LIN {X 0,Y 457.388,Z 987.215,A -85,B 0,C 180,E1 20807.693,E2 20807.693} C_VEL
LIN {X 0,Y 456.712,Z 996.163,A -85,B 0,C 180,E1 20804.974,E2 20804.974} C_VEL
LIN {X 0,Y 456.27,Z 1003.644,A -85,B 0,C 180,E1 20802.148,E2 20802.148} C_VEL
LIN {X 0,Y 456.039,Z 1009.592,A -85,B 0,C 180,E1 20799.341,E2 20799.341} C_VEL
LIN {X 0,Y 455.943,Z 1013.795,A -85,B 0,C 180,E1 20796.551,E2 20796.551} C_VEL
LIN {X 0,Y 455.903,Z 1016.656,A -85,B 0,C 180,E1 20793.742,E2 20793.742} C_VEL
LIN {X 0,Y 455.893,Z 1017.826,A -85,B 0,C 180,E1 20791.009,E2 20791.009} C_VEL
LIN {X 0,Y 455.907,Z 1017.736,A -85,B 0,C 180,E1 20788.496,E2 20788.496} C_VEL
LIN {X 0,Y 455.909,Z 1016.072,A -85,B 0,C 180,E1 20785.602,E2 20785.602} C_VEL
LIN {X 0,Y 455.929,Z 1013.325,A -85,B 0,C 180,E1 20783.076,E2 20783.076} C_VEL
LIN {X 0,Y 456.047,Z 1008.599,A -85,B 0,C 180,E1 20780.158,E2 20780.158} C_VEL
LIN {X 0,Y 456.296,Z 1003.055,A -85,B 0,C 180,E1 20777.604,E2 20777.604} C_VEL
LIN {X 0,Y 456.792,Z 994.972,A -85,B 0,C 180,E1 20774.646,E2 20774.646} C_VEL
LIN {X 0,Y 457.469,Z 986.329,A -85,B 0,C 180,E1 20772.056,E2 20772.056} C_VEL
LIN {X 0,Y 458.569,Z 974.886,A -85,B 0,C 180,E1 20769.187,E2 20769.187} C_VEL
LIN {X 0,Y 460.023,Z 962.424,A -85,B 0,C 180,E1 20766.521,E2 20766.521} C_VEL
LIN {X 0,Y 461.834,Z 948.138,A -85,B 0,C 180,E1 20763.934,E2 20763.934} C_VEL
LIN {X 0,Y 464.101,Z 931.678,A -85,B 0,C 180,E1 20761.362,E2 20761.362} C_VEL
LIN {X 0,Y 466.447,Z 915.587,A -85,B 0,C 180,E1 20759.188,E2 20759.188} C_VEL
LIN {X 0,Y 468.959,Z 897.775,A -85,B 0,C 180,E1 20757.143,E2 20757.143} C_VEL
LIN {X 0,Y 471.666,Z 878.661,A -85,B 0,C 180,E1 20755.239,E2 20755.239} C_VEL
LIN {X 0,Y 474.239,Z 859.314,A -85,B 0,C 180,E1 20753.601,E2 20753.601} C_VEL
LIN {X 0,Y 477.014,Z 837.668,A -85,B 0,C 180,E1 20752.04,E2 20752.04} C_VEL
LIN {X 0,Y 479.232,Z 818.477,A -85,B 0,C 180,E1 20750.881,E2 20750.881} C_VEL
LIN {X 0,Y 481.541,Z 795.78,A -85,B 0,C 180,E1 20749.746,E2 20749.746} C_VEL
LIN {X 0,Y 483.409,Z 774.499,A -85,B 0,C 180,E1 20748.904,E2 20748.904} C_VEL
LIN {X 0,Y 485.034,Z 751.209,A -85,B 0,C 180,E1 20748.211,E2 20748.211} C_VEL
LIN {X 0,Y 486.068,Z 729.261,A -85,B 0,C 180,E1 20747.744,E2 20747.744} C_VEL
LIN {X 0,Y 491.465,Z 519.393,A -85,B 0,C 180,E1 20744.134,E2 20744.134} C_VEL
LIN {X 0,Y 493.764,Z 431.768,A -85,B 0,C 180,E1 20742.579,E2 20742.579} C_VEL
LIN {X 0,Y 480.7,Z 411.514,A -85,B 0,C 180,E1 20740.427,E2 20740.427} C_VEL
LIN {X 0,Y 467.612,Z 392.787,A -85,B 0,C 180,E1 20738.088,E2 20738.088} C_VEL
LIN {X 0,Y 463.575,Z 387.235,A -85,B 0,C 180,E1 20737.305,E2 20737.305} C_VEL
LIN {X 0,Y 460.808,Z 382.127,A -85,B 0,C 180,E1 20736.324,E2 20736.324} C_VEL
LIN {X 0,Y 458.868,Z 378.314,A -85,B 0,C 180,E1 20735.575,E2 20735.575} C_VEL
LIN {X 0,Y 457.218,Z 375.201,A -85,B 0,C 180,E1 20734.919,E2 20734.919} C_VEL
LIN {X 0,Y 457.037,Z 374.285,A -85,B 0,C 180,E1 20734.666,E2 20734.666} C_VEL
LIN {X 0,Y 456.993,Z 374.082,A -85,B 0,C 180,E1 20731.087,E2 20731.087} C_VEL
LIN {X 0,Y 457.031,Z 374.12,A -85,B 0,C 180,E1 20727.632,E2 20727.632} C_VEL
LIN {X 0,Y 457.038,Z 374.112,A -85,B 0,C 180,E1 20724.01,E2 20724.01} C_VEL
LIN {X 0,Y 456.998,Z 374.114,A -85,B 0,C 180,E1 20720.491,E2 20720.491} C_VEL
LIN {X 0,Y 457.001,Z 374.12,A -85,B 0,C 180,E1 20716.786,E2 20716.786} C_VEL
LIN {X 0,Y 457.043,Z 374.118,A -85,B 0,C 180,E1 20713.243,E2 20713.243} C_VEL
LIN {X 0,Y 457.048,Z 374.113,A -85,B 0,C 180,E1 20709.57,E2 20709.57} C_VEL
LIN {X 0,Y 457.01,Z 374.116,A -85,B 0,C 180,E1 20706.028,E2 20706.028} C_VEL
LIN {X 0,Y 457.01,Z 374.11,A -85,B 0,C 180,E1 20702.382,E2 20702.382} C_VEL
LIN {X 0,Y 457.057,Z 374.107,A -85,B 0,C 180,E1 20698.871,E2 20698.871} C_VEL
LIN {X 0,Y 457.05,Z 374.108,A -85,B 0,C 180,E1 20695.231,E2 20695.231} C_VEL
LIN {X 0,Y 457.017,Z 374.108,A -85,B 0,C 180,E1 20691.697,E2 20691.697} C_VEL
LIN {X 0,Y 457.021,Z 374.113,A -85,B 0,C 180,E1 20687.912,E2 20687.912} C_VEL
LIN {X 0,Y 457.061,Z 374.111,A -85,B 0,C 180,E1 20684.39,E2 20684.39} C_VEL
LIN {X 0,Y 457.067,Z 374.11,A -85,B 0,C 180,E1 20680.711,E2 20680.711} C_VEL
LIN {X 0,Y 457.039,Z 374.113,A -85,B 0,C 180,E1 20677.06,E2 20677.06} C_VEL
LIN {X 0,Y 457.03,Z 374.116,A -85,B 0,C 180,E1 20673.353,E2 20673.353} C_VEL
LIN {X 0,Y 457.054,Z 374.113,A -85,B 0,C 180,E1 20669.769,E2 20669.769} C_VEL
LIN {X 0,Y 457.078,Z 374.109,A -85,B 0,C 180,E1 20666.095,E2 20666.095} C_VEL
LIN {X 0,Y 457.064,Z 374.108,A -85,B 0,C 180,E1 20662.354,E2 20662.354} C_VEL
LIN {X 0,Y 457.038,Z 374.108,A -85,B 0,C 180,E1 20658.805,E2 20658.805} C_VEL
LIN {X 0,Y 457.046,Z 374.112,A -85,B 0,C 180,E1 20655.039,E2 20655.039} C_VEL
LIN {X 0,Y 457.074,Z 374.11,A -85,B 0,C 180,E1 20651.341,E2 20651.341} C_VEL
LIN {X 0,Y 457.075,Z 374.106,A -85,B 0,C 180,E1 20647.606,E2 20647.606} C_VEL
LIN {X 0,Y 457.064,Z 374.081,A -85,B 0,C 180,E1 20643.9,E2 20643.9} C_VEL
LIN {X 0,Y 457.046,Z 374.093,A -85,B 0,C 180,E1 20640.204,E2 20640.204} C_VEL
LIN {X 0,Y 457.054,Z 374.104,A -85,B 0,C 180,E1 20636.499,E2 20636.499} C_VEL
LIN {X 0,Y 457.104,Z 374.331,A -85,B 0,C 180,E1 20635.59,E2 20635.59} C_VEL
LIN {X 0,Y 457.483,Z 375.807,A -85,B 0,C 180,E1 20635.33,E2 20635.33} C_VEL
LIN {X 0,Y 459.463,Z 378.86,A -85,B 0,C 180,E1 20634.917,E2 20634.917} C_VEL
LIN {X 0,Y 461.42,Z 380.68,A -85,B 0,C 180,E1 20634.555,E2 20634.555} C_VEL
LIN {X 0,Y 463.984,Z 384.517,A -85,B 0,C 180,E1 20634.054,E2 20634.054} C_VEL
LIN {X 0,Y 465.802,Z 386.508,A -85,B 0,C 180,E1 20633.723,E2 20633.723} C_VEL
LIN {X 0,Y 469.108,Z 390.836,A -85,B 0,C 180,E1 20633.116,E2 20633.116} C_VEL
LIN {X 0,Y 478.42,Z 403.372,A -85,B 0,C 180,E1 20631.472,E2 20631.472} C_VEL
LIN {X 0,Y 488.967,Z 418.075,A -85,B 0,C 180,E1 20629.724,E2 20629.724} C_VEL
LIN {X 0,Y 490.028,Z 420.976,A -85,B 0,C 180,E1 20629.525,E2 20629.525} C_VEL
LIN {X 0,Y 490.141,Z 425.981,A -85,B 0,C 180,E1 20629.403,E2 20629.403} C_VEL
LIN {X 0,Y 487.747,Z 440.24,A -85,B 0,C 180,E1 20629.401,E2 20629.401} C_VEL
LIN {X 0,Y 487.657,Z 441.856,A -85,B 0,C 180,E1 20629.377,E2 20629.377} C_VEL
LIN {X 0,Y 481.671,Z 650.549,A -85,B 0,C 180,E1 20625.725,E2 20625.725} C_VEL
LIN {X 0,Y 479.794,Z 714.191,A -85,B 0,C 180,E1 20624.597,E2 20624.597} C_VEL
LIN {X 0,Y 478.39,Z 736.235,A -85,B 0,C 180,E1 20624.011,E2 20624.011} C_VEL
LIN {X 0,Y 476.654,Z 758.004,A -85,B 0,C 180,E1 20623.244,E2 20623.244} C_VEL
LIN {X 0,Y 474.492,Z 778.957,A -85,B 0,C 180,E1 20622.284,E2 20622.284} C_VEL
LIN {X 0,Y 472.041,Z 800.065,A -85,B 0,C 180,E1 20621.109,E2 20621.109} C_VEL
LIN {X 0,Y 469.256,Z 820.947,A -85,B 0,C 180,E1 20619.686,E2 20619.686} C_VEL
LIN {X 0,Y 466.204,Z 842.112,A -85,B 0,C 180,E1 20617.968,E2 20617.968} C_VEL
LIN {X 0,Y 463.242,Z 861.264,A -85,B 0,C 180,E1 20616.129,E2 20616.129} C_VEL
LIN {X 0,Y 460.391,Z 879.229,A -85,B 0,C 180,E1 20614.106,E2 20614.106} C_VEL
LIN {X 0,Y 457.653,Z 896.341,A -85,B 0,C 180,E1 20611.874,E2 20611.874} C_VEL
LIN {X 0,Y 455.123,Z 912.905,A -85,B 0,C 180,E1 20609.367,E2 20609.367} C_VEL
LIN {X 0,Y 452.991,Z 928.049,A -85,B 0,C 180,E1 20606.706,E2 20606.706} C_VEL
LIN {X 0,Y 451.232,Z 941.671,A -85,B 0,C 180,E1 20603.891,E2 20603.891} C_VEL
LIN {X 0,Y 449.972,Z 952.813,A -85,B 0,C 180,E1 20601.177,E2 20601.177} C_VEL
LIN {X 0,Y 449.049,Z 962.76,A -85,B 0,C 180,E1 20598.306,E2 20598.306} C_VEL
LIN {X 0,Y 448.483,Z 970.738,A -85,B 0,C 180,E1 20595.537,E2 20595.537} C_VEL
LIN {X 0,Y 448.133,Z 977.415,A -85,B 0,C 180,E1 20592.601,E2 20592.601} C_VEL
LIN {X 0,Y 447.981,Z 982.493,A -85,B 0,C 180,E1 20589.621,E2 20589.621} C_VEL
LIN {X 0,Y 447.897,Z 985.857,A -85,B 0,C 180,E1 20586.723,E2 20586.723} C_VEL
LIN {X 0,Y 447.888,Z 987.555,A -85,B 0,C 180,E1 20584.049,E2 20584.049} C_VEL
LIN {X 0,Y 447.91,Z 987.88,A -85,B 0,C 180,E1 20581.169,E2 20581.169} C_VEL
LIN {X 0,Y 447.909,Z 986.719,A -85,B 0,C 180,E1 20578.267,E2 20578.267} C_VEL
LIN {X 0,Y 447.936,Z 984.049,A -85,B 0,C 180,E1 20575.454,E2 20575.454} C_VEL
LIN {X 0,Y 448.052,Z 979.57,A -85,B 0,C 180,E1 20572.464,E2 20572.464} C_VEL
LIN {X 0,Y 448.304,Z 973.504,A -85,B 0,C 180,E1 20569.512,E2 20569.512} C_VEL
LIN {X 0,Y 448.79,Z 966.054,A -85,B 0,C 180,E1 20566.667,E2 20566.667} C_VEL
LIN {X 0,Y 449.539,Z 957.052,A -85,B 0,C 180,E1 20563.89,E2 20563.89} C_VEL
LIN {X 0,Y 450.685,Z 946.027,A -85,B 0,C 180,E1 20561.032,E2 20561.032} C_VEL
LIN {X 0,Y 452.23,Z 933.522,A -85,B 0,C 180,E1 20558.286,E2 20558.286} C_VEL
LIN {X 0,Y 454.16,Z 919.615,A -85,B 0,C 180,E1 20555.668,E2 20555.668} C_VEL
LIN {X 0,Y 456.632,Z 903.032,A -85,B 0,C 180,E1 20553.001,E2 20553.001} C_VEL
LIN {X 0,Y 459.267,Z 886.37,A -85,B 0,C 180,E1 20550.686,E2 20550.686} C_VEL
LIN {X 0,Y 462.142,Z 868.444,A -85,B 0,C 180,E1 20548.547,E2 20548.547} C_VEL
LIN {X 0,Y 465.202,Z 848.965,A -85,B 0,C 180,E1 20546.555,E2 20546.555} C_VEL
LIN {X 0,Y 468.061,Z 829.672,A -85,B 0,C 180,E1 20544.887,E2 20544.887} C_VEL
LIN {X 0,Y 471.021,Z 808.171,A -85,B 0,C 180,E1 20543.322,E2 20543.322} C_VEL
LIN {X 0,Y 473.405,Z 788.946,A -85,B 0,C 180,E1 20542.149,E2 20542.149} C_VEL
LIN {X 0,Y 475.719,Z 767.129,A -85,B 0,C 180,E1 20541.058,E2 20541.058} C_VEL
LIN {X 0,Y 477.718,Z 745.192,A -85,B 0,C 180,E1 20540.186,E2 20540.186} C_VEL
LIN {X 0,Y 479.228,Z 723.054,A -85,B 0,C 180,E1 20539.533,E2 20539.533} C_VEL
LIN {X 0,Y 480.309,Z 699.745,A -85,B 0,C 180,E1 20539.041,E2 20539.041} C_VEL
LIN {X 0,Y 486.203,Z 492.347,A -85,B 0,C 180,E1 20535.419,E2 20535.419} C_VEL
LIN {X 0,Y 488.107,Z 428.574,A -85,B 0,C 180,E1 20534.261,E2 20534.261} C_VEL
LIN {X 0,Y 476.707,Z 412.081,A -85,B 0,C 180,E1 20532.292,E2 20532.292} C_VEL
LIN {X 0,Y 468.825,Z 401.437,A -85,B 0,C 180,E1 20530.818,E2 20530.818} C_VEL
LIN {X 0,Y 465.589,Z 397.118,A -85,B 0,C 180,E1 20530.174,E2 20530.174} C_VEL
LIN {X 0,Y 461.719,Z 392.083,A -85,B 0,C 180,E1 20529.379,E2 20529.379} C_VEL
LIN {X 0,Y 458.545,Z 387.858,A -85,B 0,C 180,E1 20528.701,E2 20528.701} C_VEL
LIN {X 0,Y 454.704,Z 383.417,A -85,B 0,C 180,E1 20527.852,E2 20527.852} C_VEL
LIN {X 0,Y 453.422,Z 381.236,A -85,B 0,C 180,E1 20527.54,E2 20527.54} C_VEL
LIN {X 0,Y 450.618,Z 378.846,A -85,B 0,C 180,E1 20526.914,E2 20526.914} C_VEL
LIN {X 0,Y 449.296,Z 376.022,A -85,B 0,C 180,E1 20526.517,E2 20526.517} C_VEL
LIN {X 0,Y 449.14,Z 375.145,A -85,B 0,C 180,E1 20526.135,E2 20526.135} C_VEL
LIN {X 0,Y 449.13,Z 375.094,A -85,B 0,C 180,E1 20522.297,E2 20522.297} C_VEL
LIN {X 0,Y 449.132,Z 375.104,A -85,B 0,C 180,E1 20518.597,E2 20518.597} C_VEL
LIN {X 0,Y 449.129,Z 375.095,A -85,B 0,C 180,E1 20514.892,E2 20514.892} C_VEL
LIN {X 0,Y 449.11,Z 375.105,A -85,B 0,C 180,E1 20511.293,E2 20511.293} C_VEL
LIN {X 0,Y 449.11,Z 375.104,A -85,B 0,C 180,E1 20507.529,E2 20507.529} C_VEL
LIN {X 0,Y 449.127,Z 375.105,A -85,B 0,C 180,E1 20503.843,E2 20503.843} C_VEL
LIN {X 0,Y 449.138,Z 375.096,A -85,B 0,C 180,E1 20500.087,E2 20500.087} C_VEL
LIN {X 0,Y 449.106,Z 375.095,A -85,B 0,C 180,E1 20496.515,E2 20496.515} C_VEL
LIN {X 0,Y 449.083,Z 375.101,A -85,B 0,C 180,E1 20492.844,E2 20492.844} C_VEL
LIN {X 0,Y 449.078,Z 375.107,A -85,B 0,C 180,E1 20489.049,E2 20489.049} C_VEL
LIN {X 0,Y 449.114,Z 375.407,A -85,B 0,C 180,E1 20486.905,E2 20486.905} C_VEL
LIN {X 0,Y 450.522,Z 378.747,A -85,B 0,C 180,E1 20486.105,E2 20486.105} C_VEL
LIN {X 0,Y 451.811,Z 380.403,A -85,B 0,C 180,E1 20485.638,E2 20485.638} C_VEL
LIN {X 0,Y 453.49,Z 383.976,A -85,B 0,C 180,E1 20484.869,E2 20484.869} C_VEL
LIN {X 0,Y 455.261,Z 386.404,A -85,B 0,C 180,E1 20484.409,E2 20484.409} C_VEL
LIN {X 0,Y 463.169,Z 397.175,A -85,B 0,C 180,E1 20482.695,E2 20482.695} C_VEL
LIN {X 0,Y 472.136,Z 410.094,A -85,B 0,C 180,E1 20480.91,E2 20480.91} C_VEL
LIN {X 0,Y 482.787,Z 426.603,A -85,B 0,C 180,E1 20478.966,E2 20478.966} C_VEL
LIN {X 0,Y 488.335,Z 435.911,A -85,B 0,C 180,E1 20478.017,E2 20478.017} C_VEL
LIN {X 0,Y 482.34,Z 638.533,A -85,B 0,C 180,E1 20474.438,E2 20474.438} C_VEL
LIN {X 0,Y 479.526,Z 739.163,A -85,B 0,C 180,E1 20472.679,E2 20472.679} C_VEL
LIN {X 0,Y 478.027,Z 762.384,A -85,B 0,C 180,E1 20472.086,E2 20472.086} C_VEL
LIN {X 0,Y 476.191,Z 785.264,A -85,B 0,C 180,E1 20471.29,E2 20471.29} C_VEL
LIN {X 0,Y 474.079,Z 805.95,A -85,B 0,C 180,E1 20470.355,E2 20470.355} C_VEL
LIN {X 0,Y 471.772,Z 826.309,A -85,B 0,C 180,E1 20469.247,E2 20469.247} C_VEL
LIN {X 0,Y 469.076,Z 847.044,A -85,B 0,C 180,E1 20467.874,E2 20467.874} C_VEL
LIN {X 0,Y 466.295,Z 867.604,A -85,B 0,C 180,E1 20466.27,E2 20466.27} C_VEL
LIN {X 0,Y 463.565,Z 886.173,A -85,B 0,C 180,E1 20464.562,E2 20464.562} C_VEL
LIN {X 0,Y 460.689,Z 905.523,A -85,B 0,C 180,E1 20462.503,E2 20462.503} C_VEL
LIN {X 0,Y 458.231,Z 921.98,A -85,B 0,C 180,E1 20460.472,E2 20460.472} C_VEL
LIN {X 0,Y 455.93,Z 937.422,A -85,B 0,C 180,E1 20458.277,E2 20458.277} C_VEL
LIN {X 0,Y 453.922,Z 951.172,A -85,B 0,C 180,E1 20456.001,E2 20456.001} C_VEL
LIN {X 0,Y 452.029,Z 965.155,A -85,B 0,C 180,E1 20453.328,E2 20453.328} C_VEL
LIN {X 0,Y 450.586,Z 977.139,A -85,B 0,C 180,E1 20450.663,E2 20450.663} C_VEL
LIN {X 0,Y 449.491,Z 987.673,A -85,B 0,C 180,E1 20447.88,E2 20447.88} C_VEL
LIN {X 0,Y 448.769,Z 996.559,A -85,B 0,C 180,E1 20445.114,E2 20445.114} C_VEL
LIN {X 0,Y 448.305,Z 1003.687,A -85,B 0,C 180,E1 20442.348,E2 20442.348} C_VEL
LIN {X 0,Y 448.046,Z 1009.649,A -85,B 0,C 180,E1 20439.475,E2 20439.475} C_VEL
LIN {X 0,Y 447.94,Z 1013.828,A -85,B 0,C 180,E1 20436.642,E2 20436.642} C_VEL
LIN {X 0,Y 447.905,Z 1016.677,A -85,B 0,C 180,E1 20433.775,E2 20433.775} C_VEL
LIN {X 0,Y 447.894,Z 1017.826,A -85,B 0,C 180,E1 20431.027,E2 20431.027} C_VEL
LIN {X 0,Y 447.907,Z 1017.736,A -85,B 0,C 180,E1 20428.469,E2 20428.469} C_VEL
LIN {X 0,Y 447.908,Z 1016.072,A -85,B 0,C 180,E1 20425.523,E2 20425.523} C_VEL
LIN {X 0,Y 447.93,Z 1013.325,A -85,B 0,C 180,E1 20422.952,E2 20422.952} C_VEL
LIN {X 0,Y 448.063,Z 1008.599,A -85,B 0,C 180,E1 20419.981,E2 20419.981} C_VEL
LIN {X 0,Y 448.338,Z 1003.055,A -85,B 0,C 180,E1 20417.38,E2 20417.38} C_VEL
LIN {X 0,Y 448.879,Z 994.971,A -85,B 0,C 180,E1 20414.369,E2 20414.369} C_VEL
LIN {X 0,Y 449.628,Z 986.285,A -85,B 0,C 180,E1 20411.719,E2 20411.719} C_VEL
LIN {X 0,Y 450.826,Z 974.885,A -85,B 0,C 180,E1 20408.812,E2 20408.812} C_VEL
LIN {X 0,Y 452.363,Z 962.648,A -85,B 0,C 180,E1 20406.146,E2 20406.146} C_VEL
LIN {X 0,Y 454.245,Z 948.907,A -85,B 0,C 180,E1 20403.606,E2 20403.606} C_VEL
LIN {X 0,Y 456.476,Z 933.886,A -85,B 0,C 180,E1 20401.181,E2 20401.181} C_VEL
LIN {X 0,Y 458.78,Z 918.361,A -85,B 0,C 180,E1 20399.053,E2 20399.053} C_VEL
LIN {X 0,Y 461.578,Z 899.875,A -85,B 0,C 180,E1 20396.847,E2 20396.847} C_VEL
LIN {X 0,Y 464.205,Z 882.408,A -85,B 0,C 180,E1 20395.051,E2 20395.051} C_VEL
LIN {X 0,Y 467.116,Z 862.195,A -85,B 0,C 180,E1 20393.26,E2 20393.26} C_VEL
LIN {X 0,Y 469.763,Z 843.056,A -85,B 0,C 180,E1 20391.814,E2 20391.814} C_VEL
LIN {X 0,Y 472.361,Z 822.483,A -85,B 0,C 180,E1 20390.507,E2 20390.507} C_VEL
LIN {X 0,Y 474.434,Z 804.256,A -85,B 0,C 180,E1 20389.533,E2 20389.533} C_VEL
LIN {X 0,Y 476.688,Z 781.174,A -85,B 0,C 180,E1 20388.527,E2 20388.527} C_VEL
LIN {X 0,Y 478.399,Z 759.67,A -85,B 0,C 180,E1 20387.805,E2 20387.805} C_VEL
LIN {X 0,Y 479.828,Z 735.636,A -85,B 0,C 180,E1 20387.232,E2 20387.232} C_VEL
LIN {X 0,Y 485.614,Z 527.459,A -85,B 0,C 180,E1 20383.602,E2 20383.602} C_VEL
LIN {X 0,Y 488.182,Z 435.454,A -85,B 0,C 180,E1 20381.953,E2 20381.953} C_VEL
LIN {X 0,Y 476.406,Z 417.107,A -85,B 0,C 180,E1 20379.957,E2 20379.957} C_VEL
LIN {X 0,Y 463.992,Z 399.176,A -85,B 0,C 180,E1 20377.694,E2 20377.694} C_VEL
LIN {X 0,Y 455.028,Z 386.96,A -85,B 0,C 180,E1 20375.922,E2 20375.922} C_VEL
LIN {X 0,Y 453.441,Z 383.956,A -85,B 0,C 180,E1 20375.337,E2 20375.337} C_VEL
LIN {X 0,Y 450.759,Z 379.042,A -85,B 0,C 180,E1 20374.292,E2 20374.292} C_VEL
LIN {X 0,Y 449.099,Z 375.317,A -85,B 0,C 180,E1 20373.456,E2 20373.456} C_VEL
LIN {X 0,Y 449.116,Z 375.058,A -85,B 0,C 180,E1 20370.012,E2 20370.012} C_VEL
LIN {X 0,Y 449.067,Z 375.101,A -85,B 0,C 180,E1 20366.442,E2 20366.442} C_VEL
LIN {X 0,Y 449.056,Z 375.103,A -85,B 0,C 180,E1 20362.794,E2 20362.794} C_VEL
LIN {X 0,Y 449.082,Z 375.11,A -85,B 0,C 180,E1 20359.239,E2 20359.239} C_VEL
LIN {X 0,Y 449.12,Z 375.098,A -85,B 0,C 180,E1 20355.494,E2 20355.494} C_VEL
LIN {X 0,Y 449.091,Z 375.099,A -85,B 0,C 180,E1 20351.819,E2 20351.819} C_VEL
LIN {X 0,Y 449.065,Z 375.1,A -85,B 0,C 180,E1 20348.192,E2 20348.192} C_VEL
LIN {X 0,Y 449.073,Z 375.107,A -85,B 0,C 180,E1 20344.469,E2 20344.469} C_VEL
LIN {X 0,Y 449.113,Z 375.106,A -85,B 0,C 180,E1 20340.892,E2 20340.892} C_VEL
LIN {X 0,Y 449.119,Z 375.106,A -85,B 0,C 180,E1 20337.192,E2 20337.192} C_VEL
LIN {X 0,Y 449.082,Z 375.108,A -85,B 0,C 180,E1 20333.608,E2 20333.608} C_VEL
LIN {X 0,Y 449.08,Z 375.107,A -85,B 0,C 180,E1 20329.869,E2 20329.869} C_VEL
LIN {X 0,Y 449.101,Z 375.102,A -85,B 0,C 180,E1 20326.218,E2 20326.218} C_VEL
LIN {X 0,Y 449.133,Z 375.097,A -85,B 0,C 180,E1 20322.643,E2 20322.643} C_VEL
LIN {X 0,Y 449.104,Z 375.101,A -85,B 0,C 180,E1 20318.995,E2 20318.995} C_VEL
LIN {X 0,Y 449.088,Z 375.101,A -85,B 0,C 180,E1 20315.396,E2 20315.396} C_VEL
LIN {X 0,Y 449.102,Z 375.093,A -85,B 0,C 180,E1 20311.691,E2 20311.691} C_VEL
LIN {X 0,Y 449.14,Z 375.093,A -85,B 0,C 180,E1 20308.156,E2 20308.156} C_VEL
LIN {X 0,Y 449.118,Z 375.097,A -85,B 0,C 180,E1 20304.474,E2 20304.474} C_VEL
LIN {X 0,Y 449.099,Z 375.103,A -85,B 0,C 180,E1 20300.776,E2 20300.776} C_VEL
LIN {X 0,Y 449.104,Z 375.104,A -85,B 0,C 180,E1 20297.057,E2 20297.057} C_VEL
LIN {X 0,Y 449.131,Z 375.092,A -85,B 0,C 180,E1 20293.456,E2 20293.456} C_VEL
LIN {X 0,Y 449.139,Z 375.096,A -85,B 0,C 180,E1 20289.704,E2 20289.704} C_VEL
LIN {X 0,Y 449.124,Z 375.102,A -85,B 0,C 180,E1 20285.989,E2 20285.989} C_VEL
LIN {X 0,Y 449.109,Z 375.089,A -85,B 0,C 180,E1 20282.291,E2 20282.291} C_VEL
LIN {X 0,Y 449.114,Z 375.072,A -85,B 0,C 180,E1 20278.592,E2 20278.592} C_VEL
LIN {X 0,Y 449.161,Z 375.309,A -85,B 0,C 180,E1 20276.931,E2 20276.931} C_VEL
LIN {X 0,Y 449.492,Z 376.701,A -85,B 0,C 180,E1 20276.669,E2 20276.669} C_VEL
LIN {X 0,Y 451.275,Z 379.636,A -85,B 0,C 180,E1 20276.273,E2 20276.273} C_VEL
LIN {X 0,Y 453.6,Z 381.672,A -85,B 0,C 180,E1 20275.818,E2 20275.818} C_VEL
LIN {X 0,Y 456.122,Z 385.504,A -85,B 0,C 180,E1 20275.293,E2 20275.293} C_VEL
LIN {X 0,Y 458.035,Z 387.55,A -85,B 0,C 180,E1 20274.925,E2 20274.925} C_VEL
LIN {X 0,Y 461.288,Z 391.848,A -85,B 0,C 180,E1 20274.293,E2 20274.293} C_VEL
LIN {X 0,Y 471.105,Z 404.838,A -85,B 0,C 180,E1 20272.485,E2 20272.485} C_VEL
LIN {X 0,Y 482.014,Z 419.923,A -85,B 0,C 180,E1 20270.601,E2 20270.601} C_VEL
LIN {X 0,Y 488.05,Z 428.946,A -85,B 0,C 180,E1 20269.606,E2 20269.606} C_VEL
LIN {X 0,Y 487.657,Z 441.856,A -85,B 0,C 180,E1 20269.377,E2 20269.377} C_VEL
LIN {X 0,Y 486.774,Z 449.554,A -85,B 0,C 180,E1 20269.324,E2 20269.324} C_VEL
LIN {X 0,Y 481.871,Z 470.179,A -85,B 0,C 180,E1 20269.506,E2 20269.506} C_VEL
LIN {X 0,Y 481.138,Z 476.789,A -85,B 0,C 180,E1 20269.456,E2 20269.456} C_VEL
LIN {X 0,Y 474.9,Z 685.168,A -85,B 0,C 180,E1 20265.786,E2 20265.786} C_VEL
LIN {X 0,Y 473.681,Z 717.796,A -85,B 0,C 180,E1 20265.165,E2 20265.165} C_VEL
LIN {X 0,Y 472.297,Z 738.069,A -85,B 0,C 180,E1 20264.607,E2 20264.607} C_VEL
LIN {X 0,Y 470.299,Z 760.875,A -85,B 0,C 180,E1 20263.771,E2 20263.771} C_VEL
LIN {X 0,Y 468.121,Z 780.902,A -85,B 0,C 180,E1 20262.83,E2 20262.83} C_VEL
LIN {X 0,Y 465.416,Z 802.513,A -85,B 0,C 180,E1 20261.59,E2 20261.59} C_VEL
LIN {X 0,Y 462.723,Z 821.616,A -85,B 0,C 180,E1 20260.265,E2 20260.265} C_VEL
LIN {X 0,Y 459.578,Z 842.279,A -85,B 0,C 180,E1 20258.566,E2 20258.566} C_VEL
LIN {X 0,Y 456.472,Z 861.304,A -85,B 0,C 180,E1 20256.726,E2 20256.726} C_VEL
LIN {X 0,Y 453.427,Z 879.309,A -85,B 0,C 180,E1 20254.676,E2 20254.676} C_VEL
LIN {X 0,Y 450.51,Z 896.471,A -85,B 0,C 180,E1 20252.413,E2 20252.413} C_VEL
LIN {X 0,Y 447.908,Z 912.218,A -85,B 0,C 180,E1 20249.996,E2 20249.996} C_VEL
LIN {X 0,Y 445.447,Z 927.997,A -85,B 0,C 180,E1 20247.166,E2 20247.166} C_VEL
LIN {X 0,Y 443.6,Z 941.026,A -85,B 0,C 180,E1 20244.434,E2 20244.434} C_VEL
LIN {X 0,Y 442.226,Z 952.261,A -85,B 0,C 180,E1 20241.676,E2 20241.676} C_VEL
LIN {X 0,Y 441.211,Z 962.3,A -85,B 0,C 180,E1 20238.758,E2 20238.758} C_VEL
LIN {X 0,Y 440.547,Z 970.685,A -85,B 0,C 180,E1 20235.808,E2 20235.808} C_VEL
LIN {X 0,Y 440.154,Z 977.362,A -85,B 0,C 180,E1 20232.82,E2 20232.82} C_VEL
LIN {X 0,Y 439.984,Z 982.422,A -85,B 0,C 180,E1 20229.809,E2 20229.809} C_VEL
LIN {X 0,Y 439.904,Z 985.83,A -85,B 0,C 180,E1 20226.842,E2 20226.842} C_VEL
LIN {X 0,Y 439.889,Z 987.538,A -85,B 0,C 180,E1 20224.122,E2 20224.122} C_VEL
LIN {X 0,Y 439.909,Z 987.885,A -85,B 0,C 180,E1 20221.19,E2 20221.19} C_VEL
LIN {X 0,Y 439.909,Z 986.816,A -85,B 0,C 180,E1 20218.326,E2 20218.326} C_VEL
LIN {X 0,Y 439.941,Z 984.072,A -85,B 0,C 180,E1 20215.359,E2 20215.359} C_VEL
LIN {X 0,Y 440.064,Z 979.622,A -85,B 0,C 180,E1 20212.321,E2 20212.321} C_VEL
LIN {X 0,Y 440.342,Z 973.597,A -85,B 0,C 180,E1 20209.324,E2 20209.324} C_VEL
LIN {X 0,Y 440.871,Z 966.121,A -85,B 0,C 180,E1 20206.41,E2 20206.41} C_VEL
LIN {X 0,Y 441.691,Z 957.124,A -85,B 0,C 180,E1 20203.579,E2 20203.579} C_VEL
LIN {X 0,Y 442.936,Z 946.099,A -85,B 0,C 180,E1 20200.667,E2 20200.667} C_VEL
LIN {X 0,Y 444.605,Z 933.597,A -85,B 0,C 180,E1 20197.871,E2 20197.871} C_VEL
LIN {X 0,Y 446.783,Z 919.178,A -85,B 0,C 180,E1 20195.11,E2 20195.11} C_VEL
LIN {X 0,Y 449.385,Z 903.427,A -85,B 0,C 180,E1 20192.511,E2 20192.511} C_VEL
LIN {X 0,Y 452.243,Z 886.493,A -85,B 0,C 180,E1 20190.124,E2 20190.124} C_VEL
LIN {X 0,Y 455.245,Z 868.873,A -85,B 0,C 180,E1 20188,E2 20188} C_VEL
LIN {X 0,Y 458.349,Z 850.337,A -85,B 0,C 180,E1 20186.069,E2 20186.069} C_VEL
LIN {X 0,Y 461.327,Z 831.286,A -85,B 0,C 180,E1 20184.393,E2 20184.393} C_VEL
LIN {X 0,Y 464.474,Z 809.871,A -85,B 0,C 180,E1 20182.798,E2 20182.798} C_VEL
LIN {X 0,Y 466.975,Z 790.764,A -85,B 0,C 180,E1 20181.61,E2 20181.61} C_VEL
LIN {X 0,Y 469.571,Z 767.813,A -85,B 0,C 180,E1 20180.439,E2 20180.439} C_VEL
LIN {X 0,Y 471.653,Z 746.082,A -85,B 0,C 180,E1 20179.565,E2 20179.565} C_VEL
LIN {X 0,Y 473.267,Z 723.764,A -85,B 0,C 180,E1 20178.897,E2 20178.897} C_VEL
LIN {X 0,Y 474.406,Z 700.716,A -85,B 0,C 180,E1 20178.402,E2 20178.402} C_VEL
LIN {X 0,Y 480.689,Z 494.451,A -85,B 0,C 180,E1 20174.756,E2 20174.756} C_VEL
LIN {X 0,Y 482.655,Z 432.375,A -85,B 0,C 180,E1 20173.615,E2 20173.615} C_VEL
LIN {X 0,Y 470.141,Z 414.244,A -85,B 0,C 180,E1 20171.35,E2 20171.35} C_VEL
LIN {X 0,Y 461.919,Z 403.31,A -85,B 0,C 180,E1 20169.721,E2 20169.721} C_VEL
LIN {X 0,Y 458.231,Z 398.502,A -85,B 0,C 180,E1 20168.944,E2 20168.944} C_VEL
LIN {X 0,Y 454.411,Z 393.527,A -85,B 0,C 180,E1 20168.096,E2 20168.096} C_VEL
LIN {X 0,Y 451.26,Z 389.54,A -85,B 0,C 180,E1 20167.368,E2 20167.368} C_VEL
LIN {X 0,Y 450.326,Z 388.205,A -85,B 0,C 180,E1 20167.143,E2 20167.143} C_VEL
LIN {X 0,Y 447.231,Z 385.014,A -85,B 0,C 180,E1 20166.419,E2 20166.419} C_VEL
LIN {X 0,Y 445.901,Z 382.445,A -85,B 0,C 180,E1 20166.05,E2 20166.05} C_VEL
LIN {X 0,Y 442.839,Z 380.034,A -85,B 0,C 180,E1 20165.294,E2 20165.294} C_VEL
LIN {X 0,Y 441.351,Z 376.979,A -85,B 0,C 180,E1 20164.809,E2 20164.809} C_VEL
LIN {X 0,Y 441.194,Z 376.113,A -85,B 0,C 180,E1 20164.302,E2 20164.302} C_VEL
LIN {X 0,Y 441.19,Z 376.084,A -85,B 0,C 180,E1 20160.52,E2 20160.52} C_VEL
LIN {X 0,Y 441.193,Z 376.081,A -85,B 0,C 180,E1 20156.753,E2 20156.753} C_VEL
LIN {X 0,Y 441.187,Z 376.093,A -85,B 0,C 180,E1 20152.971,E2 20152.971} C_VEL
LIN {X 0,Y 441.169,Z 376.092,A -85,B 0,C 180,E1 20149.29,E2 20149.29} C_VEL
LIN {X 0,Y 441.171,Z 376.095,A -85,B 0,C 180,E1 20145.564,E2 20145.564} C_VEL
LIN {X 0,Y 441.194,Z 376.092,A -85,B 0,C 180,E1 20141.913,E2 20141.913} C_VEL
LIN {X 0,Y 441.207,Z 376.088,A -85,B 0,C 180,E1 20138.043,E2 20138.043} C_VEL
LIN {X 0,Y 441.182,Z 376.085,A -85,B 0,C 180,E1 20134.207,E2 20134.207} C_VEL
LIN {X 0,Y 441.14,Z 376.086,A -85,B 0,C 180,E1 20130.688,E2 20130.688} C_VEL
LIN {X 0,Y 441.187,Z 376.396,A -85,B 0,C 180,E1 20128.492,E2 20128.492} C_VEL
LIN {X 0,Y 442.885,Z 380.136,A -85,B 0,C 180,E1 20127.5,E2 20127.5} C_VEL
LIN {X 0,Y 444.099,Z 381.894,A -85,B 0,C 180,E1 20126.986,E2 20126.986} C_VEL
LIN {X 0,Y 445.977,Z 385.156,A -85,B 0,C 180,E1 20126.298,E2 20126.298} C_VEL
LIN {X 0,Y 448.071,Z 387.766,A -85,B 0,C 180,E1 20125.783,E2 20125.783} C_VEL
LIN {X 0,Y 452.441,Z 393.552,A -85,B 0,C 180,E1 20124.737,E2 20124.737} C_VEL
LIN {X 0,Y 459.988,Z 403.937,A -85,B 0,C 180,E1 20123.058,E2 20123.058} C_VEL
LIN {X 0,Y 469.163,Z 417.43,A -85,B 0,C 180,E1 20121.184,E2 20121.184} C_VEL
LIN {X 0,Y 480.342,Z 435.102,A -85,B 0,C 180,E1 20119.108,E2 20119.108} C_VEL
LIN {X 0,Y 482.867,Z 439.645,A -85,B 0,C 180,E1 20118.658,E2 20118.658} C_VEL
LIN {X 0,Y 476.5,Z 641.209,A -85,B 0,C 180,E1 20115.059,E2 20115.059} C_VEL
LIN {X 0,Y 473.563,Z 739.133,A -85,B 0,C 180,E1 20113.324,E2 20113.324} C_VEL
LIN {X 0,Y 471.954,Z 762.476,A -85,B 0,C 180,E1 20112.722,E2 20112.722} C_VEL
LIN {X 0,Y 470,Z 785.356,A -85,B 0,C 180,E1 20111.915,E2 20111.915} C_VEL
LIN {X 0,Y 467.777,Z 805.975,A -85,B 0,C 180,E1 20110.973,E2 20110.973} C_VEL
LIN {X 0,Y 465.272,Z 826.811,A -85,B 0,C 180,E1 20109.824,E2 20109.824} C_VEL
LIN {X 0,Y 462.422,Z 847.413,A -85,B 0,C 180,E1 20108.439,E2 20108.439} C_VEL
LIN {X 0,Y 459.38,Z 868.407,A -85,B 0,C 180,E1 20106.769,E2 20106.769} C_VEL
LIN {X 0,Y 456.593,Z 886.36,A -85,B 0,C 180,E1 20105.091,E2 20105.091} C_VEL
LIN {X 0,Y 453.448,Z 906.097,A -85,B 0,C 180,E1 20102.949,E2 20102.949} C_VEL
LIN {X 0,Y 450.841,Z 922.566,A -85,B 0,C 180,E1 20100.878,E2 20100.878} C_VEL
LIN {X 0,Y 448.265,Z 938.906,A -85,B 0,C 180,E1 20098.501,E2 20098.501} C_VEL
LIN {X 0,Y 446.22,Z 952.711,A -85,B 0,C 180,E1 20096.198,E2 20096.198} C_VEL
LIN {X 0,Y 444.22,Z 966.423,A -85,B 0,C 180,E1 20093.481,E2 20093.481} C_VEL
LIN {X 0,Y 442.705,Z 978.253,A -85,B 0,C 180,E1 20090.769,E2 20090.769} C_VEL
LIN {X 0,Y 441.554,Z 988.589,A -85,B 0,C 180,E1 20087.94,E2 20087.94} C_VEL
LIN {X 0,Y 440.726,Z 997.983,A -85,B 0,C 180,E1 20084.858,E2 20084.858} C_VEL
LIN {X 0,Y 440.298,Z 1004.552,A -85,B 0,C 180,E1 20082.196,E2 20082.196} C_VEL
LIN {X 0,Y 440.042,Z 1010.423,A -85,B 0,C 180,E1 20079.156,E2 20079.156} C_VEL
LIN {X 0,Y 439.945,Z 1014.114,A -85,B 0,C 180,E1 20076.529,E2 20076.529} C_VEL
LIN {X 0,Y 439.892,Z 1016.846,A -85,B 0,C 180,E1 20073.522,E2 20073.522} C_VEL
LIN {X 0,Y 439.889,Z 1017.848,A -85,B 0,C 180,E1 20070.916,E2 20070.916} C_VEL
LIN {X 0,Y 439.909,Z 1017.66,A -85,B 0,C 180,E1 20068.05,E2 20068.05} C_VEL
LIN {X 0,Y 439.91,Z 1015.844,A -85,B 0,C 180,E1 20065.18,E2 20065.18} C_VEL
LIN {X 0,Y 439.967,Z 1012.686,A -85,B 0,C 180,E1 20062.299,E2 20062.299} C_VEL
LIN {X 0,Y 440.131,Z 1007.836,A -85,B 0,C 180,E1 20059.401,E2 20059.401} C_VEL
LIN {X 0,Y 440.487,Z 1001.528,A -85,B 0,C 180,E1 20056.484,E2 20056.484} C_VEL
LIN {X 0,Y 441.066,Z 993.755,A -85,B 0,C 180,E1 20053.679,E2 20053.679} C_VEL
LIN {X 0,Y 441.994,Z 984.459,A -85,B 0,C 180,E1 20050.857,E2 20050.857} C_VEL
LIN {X 0,Y 443.247,Z 973.736,A -85,B 0,C 180,E1 20048.154,E2 20048.154} C_VEL
LIN {X 0,Y 444.948,Z 961.269,A -85,B 0,C 180,E1 20045.441,E2 20045.441} C_VEL
LIN {X 0,Y 446.778,Z 948.862,A -85,B 0,C 180,E1 20043.129,E2 20043.129} C_VEL
LIN {X 0,Y 449.187,Z 933.255,A -85,B 0,C 180,E1 20040.623,E2 20040.623} C_VEL
LIN {X 0,Y 451.762,Z 916.967,A -85,B 0,C 180,E1 20038.369,E2 20038.369} C_VEL
LIN {X 0,Y 454.822,Z 898.07,A -85,B 0,C 180,E1 20036.115,E2 20036.115} C_VEL
LIN {X 0,Y 457.712,Z 879.987,A -85,B 0,C 180,E1 20034.25,E2 20034.25} C_VEL
LIN {X 0,Y 460.738,Z 860.144,A -85,B 0,C 180,E1 20032.51,E2 20032.51} C_VEL
LIN {X 0,Y 463.716,Z 839.852,A -85,B 0,C 180,E1 20030.986,E2 20030.986} C_VEL
LIN {X 0,Y 466.454,Z 818.606,A -85,B 0,C 180,E1 20029.665,E2 20029.665} C_VEL
LIN {X 0,Y 469.043,Z 796.277,A -85,B 0,C 180,E1 20028.522,E2 20028.522} C_VEL
LIN {X 0,Y 471.13,Z 775.083,A -85,B 0,C 180,E1 20027.665,E2 20027.665} C_VEL
LIN {X 0,Y 472.991,Z 751.564,A -85,B 0,C 180,E1 20026.945,E2 20026.945} C_VEL
LIN {X 0,Y 474.14,Z 729.857,A -85,B 0,C 180,E1 20026.471,E2 20026.471} C_VEL
LIN {X 0,Y 480.299,Z 519.471,A -85,B 0,C 180,E1 20022.774,E2 20022.774} C_VEL
LIN {X 0,Y 482.692,Z 439.246,A -85,B 0,C 180,E1 20021.319,E2 20021.319} C_VEL
LIN {X 0,Y 472.156,Z 422.69,A -85,B 0,C 180,E1 20019.48,E2 20019.48} C_VEL
LIN {X 0,Y 460.256,Z 405.397,A -85,B 0,C 180,E1 20017.268,E2 20017.268} C_VEL
LIN {X 0,Y 449.103,Z 390.229,A -85,B 0,C 180,E1 20015.018,E2 20015.018} C_VEL
LIN {X 0,Y 446.205,Z 385.768,A -85,B 0,C 180,E1 20014.302,E2 20014.302} C_VEL
LIN {X 0,Y 443.806,Z 381.453,A -85,B 0,C 180,E1 20013.347,E2 20013.347} C_VEL
LIN {X 0,Y 441.528,Z 377.731,A -85,B 0,C 180,E1 20012.458,E2 20012.458} C_VEL
LIN {X 0,Y 441.2,Z 376.276,A -85,B 0,C 180,E1 20012.094,E2 20012.094} C_VEL
LIN {X 0,Y 441.118,Z 376.074,A -85,B 0,C 180,E1 20008.707,E2 20008.707} C_VEL
LIN {X 0,Y 441.116,Z 376.102,A -85,B 0,C 180,E1 20004.935,E2 20004.935} C_VEL
LIN {X 0,Y 441.138,Z 376.094,A -85,B 0,C 180,E1 20001.262,E2 20001.262} C_VEL
LIN {X 0,Y 441.172,Z 376.086,A -85,B 0,C 180,E1 19997.543,E2 19997.543} C_VEL
LIN {X 0,Y 441.148,Z 376.09,A -85,B 0,C 180,E1 19993.901,E2 19993.901} C_VEL
LIN {X 0,Y 441.126,Z 376.097,A -85,B 0,C 180,E1 19990.315,E2 19990.315} C_VEL
LIN {X 0,Y 441.131,Z 376.095,A -85,B 0,C 180,E1 19986.507,E2 19986.507} C_VEL
LIN {X 0,Y 441.161,Z 376.086,A -85,B 0,C 180,E1 19982.858,E2 19982.858} C_VEL
LIN {X 0,Y 441.184,Z 376.084,A -85,B 0,C 180,E1 19979.22,E2 19979.22} C_VEL
LIN {X 0,Y 441.146,Z 376.088,A -85,B 0,C 180,E1 19975.58,E2 19975.58} C_VEL
LIN {X 0,Y 441.138,Z 376.085,A -85,B 0,C 180,E1 19971.921,E2 19971.921} C_VEL
LIN {X 0,Y 441.156,Z 376.087,A -85,B 0,C 180,E1 19968.23,E2 19968.23} C_VEL
LIN {X 0,Y 441.199,Z 376.083,A -85,B 0,C 180,E1 19964.624,E2 19964.624} C_VEL
LIN {X 0,Y 441.181,Z 376.086,A -85,B 0,C 180,E1 19960.815,E2 19960.815} C_VEL
LIN {X 0,Y 441.153,Z 376.091,A -85,B 0,C 180,E1 19957.196,E2 19957.196} C_VEL
LIN {X 0,Y 441.155,Z 376.093,A -85,B 0,C 180,E1 19953.481,E2 19953.481} C_VEL
LIN {X 0,Y 441.178,Z 376.092,A -85,B 0,C 180,E1 19949.792,E2 19949.792} C_VEL
LIN {X 0,Y 441.198,Z 376.086,A -85,B 0,C 180,E1 19946.031,E2 19946.031} C_VEL
LIN {X 0,Y 441.191,Z 376.083,A -85,B 0,C 180,E1 19942.263,E2 19942.263} C_VEL
LIN {X 0,Y 441.168,Z 376.084,A -85,B 0,C 180,E1 19938.563,E2 19938.563} C_VEL
LIN {X 0,Y 441.164,Z 376.091,A -85,B 0,C 180,E1 19934.81,E2 19934.81} C_VEL
LIN {X 0,Y 441.175,Z 376.089,A -85,B 0,C 180,E1 19931,E2 19931} C_VEL
LIN {X 0,Y 441.194,Z 376.084,A -85,B 0,C 180,E1 19927.301,E2 19927.301} C_VEL
LIN {X 0,Y 441.195,Z 376.054,A -85,B 0,C 180,E1 19923.489,E2 19923.489} C_VEL
LIN {X 0,Y 441.192,Z 376.058,A -85,B 0,C 180,E1 19919.75,E2 19919.75} C_VEL
LIN {X 0,Y 441.192,Z 376.214,A -85,B 0,C 180,E1 19918.413,E2 19918.413} C_VEL
LIN {X 0,Y 441.501,Z 377.549,A -85,B 0,C 180,E1 19918.097,E2 19918.097} C_VEL
LIN {X 0,Y 443.334,Z 380.596,A -85,B 0,C 180,E1 19917.655,E2 19917.655} C_VEL
LIN {X 0,Y 445.735,Z 382.707,A -85,B 0,C 180,E1 19917.164,E2 19917.164} C_VEL
LIN {X 0,Y 448.23,Z 386.518,A -85,B 0,C 180,E1 19916.618,E2 19916.618} C_VEL
LIN {X 0,Y 450.397,Z 388.731,A -85,B 0,C 180,E1 19916.179,E2 19916.179} C_VEL
LIN {X 0,Y 453.661,Z 393.015,A -85,B 0,C 180,E1 19915.506,E2 19915.506} C_VEL
LIN {X 0,Y 463.626,Z 406.113,A -85,B 0,C 180,E1 19913.571,E2 19913.571} C_VEL
LIN {X 0,Y 474.371,Z 420.762,A -85,B 0,C 180,E1 19911.639,E2 19911.639} C_VEL
LIN {X 0,Y 482.548,Z 432.768,A -85,B 0,C 180,E1 19910.242,E2 19910.242} C_VEL
LIN {X 0,Y 481.138,Z 476.789,A -85,B 0,C 180,E1 19909.456,E2 19909.456} C_VEL
LIN {X 0,Y 480.208,Z 484.487,A -85,B 0,C 180,E1 19909.407,E2 19909.407} C_VEL
LIN {X 0,Y 475.287,Z 505.1,A -85,B 0,C 180,E1 19909.592,E2 19909.592} C_VEL
LIN {X 0,Y 474.545,Z 511.706,A -85,B 0,C 180,E1 19909.542,E2 19909.542} C_VEL
LIN {X 0,Y 468.162,Z 711.488,A -85,B 0,C 180,E1 19905.976,E2 19905.976} C_VEL
LIN {X 0,Y 466.601,Z 735.251,A -85,B 0,C 180,E1 19905.365,E2 19905.365} C_VEL
LIN {X 0,Y 464.716,Z 756.98,A -85,B 0,C 180,E1 19904.599,E2 19904.599} C_VEL
LIN {X 0,Y 462.36,Z 778.198,A -85,B 0,C 180,E1 19903.629,E2 19903.629} C_VEL
LIN {X 0,Y 459.897,Z 797.56,A -85,B 0,C 180,E1 19902.553,E2 19902.553} C_VEL
LIN {X 0,Y 456.737,Z 819.042,A -85,B 0,C 180,E1 19901.103,E2 19901.103} C_VEL
LIN {X 0,Y 453.629,Z 838.871,A -85,B 0,C 180,E1 19899.511,E2 19899.511} C_VEL
LIN {X 0,Y 450.389,Z 857.664,A -85,B 0,C 180,E1 19897.714,E2 19897.714} C_VEL
LIN {X 0,Y 447.153,Z 875.853,A -85,B 0,C 180,E1 19895.702,E2 19895.702} C_VEL
LIN {X 0,Y 444.071,Z 892.964,A -85,B 0,C 180,E1 19893.481,E2 19893.481} C_VEL
LIN {X 0,Y 441.143,Z 909.197,A -85,B 0,C 180,E1 19891.035,E2 19891.035} C_VEL
LIN {X 0,Y 438.597,Z 923.997,A -85,B 0,C 180,E1 19888.429,E2 19888.429} C_VEL
LIN {X 0,Y 436.375,Z 938.082,A -85,B 0,C 180,E1 19885.528,E2 19885.528} C_VEL
LIN {X 0,Y 434.643,Z 950.72,A -85,B 0,C 180,E1 19882.462,E2 19882.462} C_VEL
LIN {X 0,Y 433.472,Z 961.032,A -85,B 0,C 180,E1 19879.497,E2 19879.497} C_VEL
LIN {X 0,Y 432.693,Z 969.551,A -85,B 0,C 180,E1 19876.5,E2 19876.5} C_VEL
LIN {X 0,Y 432.213,Z 976.469,A -85,B 0,C 180,E1 19873.465,E2 19873.465} C_VEL
LIN {X 0,Y 431.991,Z 981.627,A -85,B 0,C 180,E1 19870.528,E2 19870.528} C_VEL
LIN {X 0,Y 431.917,Z 985.134,A -85,B 0,C 180,E1 19867.685,E2 19867.685} C_VEL
LIN {X 0,Y 431.911,Z 987.25,A -85,B 0,C 180,E1 19864.786,E2 19864.786} C_VEL
LIN {X 0,Y 431.906,Z 987.984,A -85,B 0,C 180,E1 19861.816,E2 19861.816} C_VEL
LIN {X 0,Y 431.914,Z 987.155,A -85,B 0,C 180,E1 19858.917,E2 19858.917} C_VEL
LIN {X 0,Y 431.912,Z 984.814,A -85,B 0,C 180,E1 19855.926,E2 19855.926} C_VEL
LIN {X 0,Y 432.003,Z 981.321,A -85,B 0,C 180,E1 19853.166,E2 19853.166} C_VEL
LIN {X 0,Y 432.266,Z 975.915,A -85,B 0,C 180,E1 19850.17,E2 19850.17} C_VEL
LIN {X 0,Y 432.754,Z 968.702,A -85,B 0,C 180,E1 19847.09,E2 19847.09} C_VEL
LIN {X 0,Y 433.553,Z 960.159,A -85,B 0,C 180,E1 19844.145,E2 19844.145} C_VEL
LIN {X 0,Y 434.744,Z 949.907,A -85,B 0,C 180,E1 19841.227,E2 19841.227} C_VEL
LIN {X 0,Y 436.487,Z 937.277,A -85,B 0,C 180,E1 19838.206,E2 19838.206} C_VEL
LIN {X 0,Y 438.706,Z 923.476,A -85,B 0,C 180,E1 19835.373,E2 19835.373} C_VEL
LIN {X 0,Y 441.32,Z 908.376,A -85,B 0,C 180,E1 19832.728,E2 19832.728} C_VEL
LIN {X 0,Y 444.356,Z 891.566,A -85,B 0,C 180,E1 19830.222,E2 19830.222} C_VEL
LIN {X 0,Y 447.467,Z 874.588,A -85,B 0,C 180,E1 19828.036,E2 19828.036} C_VEL
LIN {X 0,Y 450.659,Z 856.495,A -85,B 0,C 180,E1 19826.059,E2 19826.059} C_VEL
LIN {X 0,Y 453.962,Z 837.102,A -85,B 0,C 180,E1 19824.235,E2 19824.235} C_VEL
LIN {X 0,Y 456.976,Z 817.991,A -85,B 0,C 180,E1 19822.718,E2 19822.718} C_VEL
LIN {X 0,Y 460.097,Z 796.384,A -85,B 0,C 180,E1 19821.28,E2 19821.28} C_VEL
LIN {X 0,Y 462.498,Z 777.435,A -85,B 0,C 180,E1 19820.236,E2 19820.236} C_VEL
LIN {X 0,Y 464.951,Z 754.313,A -85,B 0,C 180,E1 19819.206,E2 19819.206} C_VEL
LIN {X 0,Y 466.78,Z 732.967,A -85,B 0,C 180,E1 19818.472,E2 19818.472} C_VEL
LIN {X 0,Y 468.222,Z 709.434,A -85,B 0,C 180,E1 19817.899,E2 19817.899} C_VEL
LIN {X 0,Y 475.256,Z 496.565,A -85,B 0,C 180,E1 19814.078,E2 19814.078} C_VEL
LIN {X 0,Y 477.35,Z 436.488,A -85,B 0,C 180,E1 19812.969,E2 19812.969} C_VEL
LIN {X 0,Y 466.387,Z 420.405,A -85,B 0,C 180,E1 19810.916,E2 19810.916} C_VEL
LIN {X 0,Y 458.146,Z 409.3,A -85,B 0,C 180,E1 19809.231,E2 19809.231} C_VEL
LIN {X 0,Y 454.666,Z 404.739,A -85,B 0,C 180,E1 19808.473,E2 19808.473} C_VEL
LIN {X 0,Y 451.182,Z 400.154,A -85,B 0,C 180,E1 19807.674,E2 19807.674} C_VEL
LIN {X 0,Y 446.981,Z 394.841,A -85,B 0,C 180,E1 19806.676,E2 19806.676} C_VEL
LIN {X 0,Y 443.834,Z 390.995,A -85,B 0,C 180,E1 19805.884,E2 19805.884} C_VEL
LIN {X 0,Y 442.933,Z 389.52,A -85,B 0,C 180,E1 19805.636,E2 19805.636} C_VEL
LIN {X 0,Y 439.801,Z 386.532,A -85,B 0,C 180,E1 19804.826,E2 19804.826} C_VEL
LIN {X 0,Y 438.09,Z 383.493,A -85,B 0,C 180,E1 19804.32,E2 19804.32} C_VEL
LIN {X 0,Y 434.975,Z 381.129,A -85,B 0,C 180,E1 19803.46,E2 19803.46} C_VEL
LIN {X 0,Y 433.435,Z 378.048,A -85,B 0,C 180,E1 19802.91,E2 19802.91} C_VEL
LIN {X 0,Y 433.256,Z 377.11,A -85,B 0,C 180,E1 19802.381,E2 19802.381} C_VEL
LIN {X 0,Y 433.255,Z 377.082,A -85,B 0,C 180,E1 19798.546,E2 19798.546} C_VEL
LIN {X 0,Y 433.255,Z 377.069,A -85,B 0,C 180,E1 19794.704,E2 19794.704} C_VEL
LIN {X 0,Y 433.242,Z 377.081,A -85,B 0,C 180,E1 19790.972,E2 19790.972} C_VEL
LIN {X 0,Y 433.228,Z 377.083,A -85,B 0,C 180,E1 19787.2,E2 19787.2} C_VEL
LIN {X 0,Y 433.225,Z 377.083,A -85,B 0,C 180,E1 19783.371,E2 19783.371} C_VEL
LIN {X 0,Y 433.233,Z 377.071,A -85,B 0,C 180,E1 19779.605,E2 19779.605} C_VEL
LIN {X 0,Y 433.253,Z 377.07,A -85,B 0,C 180,E1 19775.891,E2 19775.891} C_VEL
LIN {X 0,Y 433.255,Z 377.083,A -85,B 0,C 180,E1 19772.065,E2 19772.065} C_VEL
LIN {X 0,Y 433.275,Z 377.415,A -85,B 0,C 180,E1 19770.255,E2 19770.255} C_VEL
LIN {X 0,Y 434.942,Z 381.152,A -85,B 0,C 180,E1 19769.161,E2 19769.161} C_VEL
LIN {X 0,Y 436.467,Z 383.151,A -85,B 0,C 180,E1 19768.552,E2 19768.552} C_VEL
LIN {X 0,Y 439.805,Z 387.572,A -85,B 0,C 180,E1 19767.592,E2 19767.592} C_VEL
LIN {X 0,Y 445.205,Z 394.708,A -85,B 0,C 180,E1 19766.154,E2 19766.154} C_VEL
LIN {X 0,Y 449.407,Z 400.317,A -85,B 0,C 180,E1 19765.126,E2 19765.126} C_VEL
LIN {X 0,Y 458.096,Z 412.422,A -85,B 0,C 180,E1 19763.154,E2 19763.154} C_VEL
LIN {X 0,Y 469.449,Z 429.806,A -85,B 0,C 180,E1 19760.829,E2 19760.829} C_VEL
LIN {X 0,Y 477.483,Z 443.285,A -85,B 0,C 180,E1 19759.317,E2 19759.317} C_VEL
LIN {X 0,Y 470.688,Z 644.968,A -85,B 0,C 180,E1 19755.676,E2 19755.676} C_VEL
LIN {X 0,Y 467.691,Z 738.695,A -85,B 0,C 180,E1 19753.996,E2 19753.996} C_VEL
LIN {X 0,Y 465.982,Z 762.147,A -85,B 0,C 180,E1 19753.388,E2 19753.388} C_VEL
LIN {X 0,Y 463.95,Z 784.701,A -85,B 0,C 180,E1 19752.589,E2 19752.589} C_VEL
LIN {X 0,Y 461.618,Z 805.26,A -85,B 0,C 180,E1 19751.647,E2 19751.647} C_VEL
LIN {X 0,Y 458.972,Z 826.241,A -85,B 0,C 180,E1 19750.483,E2 19750.483} C_VEL
LIN {X 0,Y 455.935,Z 847.01,A -85,B 0,C 180,E1 19749.076,E2 19749.076} C_VEL
LIN {X 0,Y 452.717,Z 867.896,A -85,B 0,C 180,E1 19747.402,E2 19747.402} C_VEL
LIN {X 0,Y 449.768,Z 885.871,A -85,B 0,C 180,E1 19745.704,E2 19745.704} C_VEL
LIN {X 0,Y 446.387,Z 905.792,A -85,B 0,C 180,E1 19743.517,E2 19743.517} C_VEL
LIN {X 0,Y 443.576,Z 922.519,A -85,B 0,C 180,E1 19741.382,E2 19741.382} C_VEL
LIN {X 0,Y 440.894,Z 938.399,A -85,B 0,C 180,E1 19739.036,E2 19739.036} C_VEL
LIN {X 0,Y 438.588,Z 953.131,A -85,B 0,C 180,E1 19736.543,E2 19736.543} C_VEL
LIN {X 0,Y 436.592,Z 966.402,A -85,B 0,C 180,E1 19733.917,E2 19733.917} C_VEL
LIN {X 0,Y 434.955,Z 978.244,A -85,B 0,C 180,E1 19731.159,E2 19731.159} C_VEL
LIN {X 0,Y 433.71,Z 988.588,A -85,B 0,C 180,E1 19728.276,E2 19728.276} C_VEL
LIN {X 0,Y 432.813,Z 997.982,A -85,B 0,C 180,E1 19725.136,E2 19725.136} C_VEL
LIN {X 0,Y 432.338,Z 1004.552,A -85,B 0,C 180,E1 19722.424,E2 19722.424} C_VEL
LIN {X 0,Y 432.051,Z 1010.423,A -85,B 0,C 180,E1 19719.326,E2 19719.326} C_VEL
LIN {X 0,Y 431.941,Z 1014.114,A -85,B 0,C 180,E1 19716.65,E2 19716.65} C_VEL
LIN {X 0,Y 431.895,Z 1016.846,A -85,B 0,C 180,E1 19713.588,E2 19713.588} C_VEL
LIN {X 0,Y 431.891,Z 1017.848,A -85,B 0,C 180,E1 19710.933,E2 19710.933} C_VEL
LIN {X 0,Y 431.907,Z 1017.69,A -85,B 0,C 180,E1 19708.147,E2 19708.147} C_VEL
LIN {X 0,Y 431.91,Z 1015.958,A -85,B 0,C 180,E1 19705.224,E2 19705.224} C_VEL
LIN {X 0,Y 431.947,Z 1013.165,A -85,B 0,C 180,E1 19702.556,E2 19702.556} C_VEL
LIN {X 0,Y 432.129,Z 1008.344,A -85,B 0,C 180,E1 19699.472,E2 19699.472} C_VEL
LIN {X 0,Y 432.462,Z 1002.683,A -85,B 0,C 180,E1 19696.742,E2 19696.742} C_VEL
LIN {X 0,Y 433.105,Z 994.564,A -85,B 0,C 180,E1 19693.646,E2 19693.646} C_VEL
LIN {X 0,Y 434.021,Z 985.867,A -85,B 0,C 180,E1 19690.911,E2 19690.911} C_VEL
LIN {X 0,Y 435.391,Z 974.881,A -85,B 0,C 180,E1 19688.023,E2 19688.023} C_VEL
LIN {X 0,Y 436.905,Z 964.222,A -85,B 0,C 180,E1 19685.618,E2 19685.618} C_VEL
LIN {X 0,Y 439.055,Z 950.09,A -85,B 0,C 180,E1 19682.911,E2 19682.911} C_VEL
LIN {X 0,Y 441.537,Z 935.032,A -85,B 0,C 180,E1 19680.407,E2 19680.407} C_VEL
LIN {X 0,Y 444.333,Z 918.324,A -85,B 0,C 180,E1 19678.031,E2 19678.031} C_VEL
LIN {X 0,Y 447.466,Z 900.292,A -85,B 0,C 180,E1 19675.806,E2 19675.806} C_VEL
LIN {X 0,Y 450.524,Z 882.137,A -85,B 0,C 180,E1 19673.884,E2 19673.884} C_VEL
LIN {X 0,Y 453.923,Z 861.381,A -85,B 0,C 180,E1 19672.007,E2 19672.007} C_VEL
LIN {X 0,Y 456.942,Z 841.935,A -85,B 0,C 180,E1 19670.513,E2 19670.513} C_VEL
LIN {X 0,Y 459.925,Z 820.441,A -85,B 0,C 180,E1 19669.136,E2 19669.136} C_VEL
LIN {X 0,Y 462.648,Z 798.755,A -85,B 0,C 180,E1 19667.985,E2 19667.985} C_VEL
LIN {X 0,Y 464.969,Z 776.396,A -85,B 0,C 180,E1 19667.059,E2 19667.059} C_VEL
LIN {X 0,Y 466.971,Z 752.989,A -85,B 0,C 180,E1 19666.32,E2 19666.32} C_VEL
LIN {X 0,Y 468.217,Z 731.065,A -85,B 0,C 180,E1 19665.829,E2 19665.829} C_VEL
LIN {X 0,Y 474.798,Z 520.557,A -85,B 0,C 180,E1 19662.087,E2 19662.087} C_VEL
LIN {X 0,Y 477.315,Z 443.079,A -85,B 0,C 180,E1 19660.679,E2 19660.679} C_VEL
LIN {X 0,Y 466.056,Z 425.409,A -85,B 0,C 180,E1 19658.652,E2 19658.652} C_VEL
LIN {X 0,Y 455.734,Z 410.548,A -85,B 0,C 180,E1 19656.676,E2 19656.676} C_VEL
LIN {X 0,Y 445.775,Z 396.779,A -85,B 0,C 180,E1 19654.608,E2 19654.608} C_VEL
LIN {X 0,Y 441.486,Z 391.088,A -85,B 0,C 180,E1 19653.662,E2 19653.662} C_VEL
LIN {X 0,Y 437.663,Z 386.025,A -85,B 0,C 180,E1 19652.781,E2 19652.781} C_VEL
LIN {X 0,Y 435.201,Z 381.422,A -85,B 0,C 180,E1 19651.743,E2 19651.743} C_VEL
LIN {X 0,Y 433.336,Z 377.917,A -85,B 0,C 180,E1 19650.881,E2 19650.881} C_VEL
LIN {X 0,Y 433.203,Z 377.127,A -85,B 0,C 180,E1 19650.515,E2 19650.515} C_VEL
LIN {X 0,Y 433.176,Z 377.082,A -85,B 0,C 180,E1 19646.898,E2 19646.898} C_VEL
LIN {X 0,Y 433.184,Z 377.077,A -85,B 0,C 180,E1 19643.103,E2 19643.103} C_VEL
LIN {X 0,Y 433.23,Z 377.08,A -85,B 0,C 180,E1 19639.551,E2 19639.551} C_VEL
LIN {X 0,Y 433.225,Z 377.082,A -85,B 0,C 180,E1 19635.782,E2 19635.782} C_VEL
LIN {X 0,Y 433.193,Z 377.079,A -85,B 0,C 180,E1 19632.124,E2 19632.124} C_VEL
LIN {X 0,Y 433.187,Z 377.076,A -85,B 0,C 180,E1 19628.361,E2 19628.361} C_VEL
LIN {X 0,Y 433.209,Z 377.079,A -85,B 0,C 180,E1 19624.766,E2 19624.766} C_VEL
LIN {X 0,Y 433.249,Z 377.078,A -85,B 0,C 180,E1 19621.057,E2 19621.057} C_VEL
LIN {X 0,Y 433.227,Z 377.083,A -85,B 0,C 180,E1 19617.354,E2 19617.354} C_VEL
LIN {X 0,Y 433.204,Z 377.086,A -85,B 0,C 180,E1 19613.639,E2 19613.639} C_VEL
LIN {X 0,Y 433.204,Z 377.085,A -85,B 0,C 180,E1 19609.897,E2 19609.897} C_VEL
LIN {X 0,Y 433.216,Z 377.08,A -85,B 0,C 180,E1 19606.111,E2 19606.111} C_VEL
LIN {X 0,Y 433.249,Z 377.071,A -85,B 0,C 180,E1 19602.402,E2 19602.402} C_VEL
LIN {X 0,Y 433.255,Z 377.07,A -85,B 0,C 180,E1 19598.615,E2 19598.615} C_VEL
LIN {X 0,Y 433.228,Z 377.073,A -85,B 0,C 180,E1 19594.87,E2 19594.87} C_VEL
LIN {X 0,Y 433.213,Z 377.073,A -85,B 0,C 180,E1 19591.159,E2 19591.159} C_VEL
LIN {X 0,Y 433.22,Z 377.081,A -85,B 0,C 180,E1 19587.311,E2 19587.311} C_VEL
LIN {X 0,Y 433.241,Z 377.082,A -85,B 0,C 180,E1 19583.621,E2 19583.621} C_VEL
LIN {X 0,Y 433.265,Z 377.074,A -85,B 0,C 180,E1 19579.797,E2 19579.797} C_VEL
LIN {X 0,Y 433.255,Z 377.07,A -85,B 0,C 180,E1 19576,E2 19576} C_VEL
LIN {X 0,Y 433.243,Z 377.075,A -85,B 0,C 180,E1 19572.182,E2 19572.182} C_VEL
LIN {X 0,Y 433.228,Z 377.082,A -85,B 0,C 180,E1 19568.519,E2 19568.519} C_VEL
LIN {X 0,Y 433.232,Z 377.051,A -85,B 0,C 180,E1 19564.747,E2 19564.747} C_VEL
LIN {X 0,Y 433.255,Z 377.069,A -85,B 0,C 180,E1 19560.967,E2 19560.967} C_VEL
LIN {X 0,Y 433.278,Z 377.277,A -85,B 0,C 180,E1 19559.892,E2 19559.892} C_VEL
LIN {X 0,Y 433.668,Z 378.759,A -85,B 0,C 180,E1 19559.566,E2 19559.566} C_VEL
LIN {X 0,Y 435.568,Z 381.74,A -85,B 0,C 180,E1 19559.087,E2 19559.087} C_VEL
LIN {X 0,Y 437.911,Z 383.791,A -85,B 0,C 180,E1 19558.574,E2 19558.574} C_VEL
LIN {X 0,Y 440.45,Z 387.611,A -85,B 0,C 180,E1 19557.985,E2 19557.985} C_VEL
LIN {X 0,Y 442.574,Z 389.769,A -85,B 0,C 180,E1 19557.534,E2 19557.534} C_VEL
LIN {X 0,Y 445.749,Z 393.976,A -85,B 0,C 180,E1 19556.849,E2 19556.849} C_VEL
LIN {X 0,Y 447.411,Z 395.95,A -85,B 0,C 180,E1 19556.502,E2 19556.502} C_VEL
LIN {X 0,Y 452.324,Z 402.418,A -85,B 0,C 180,E1 19555.482,E2 19555.482} C_VEL
LIN {X 0,Y 460.302,Z 412.881,A -85,B 0,C 180,E1 19553.917,E2 19553.917} C_VEL
LIN {X 0,Y 472.525,Z 429.696,A -85,B 0,C 180,E1 19551.691,E2 19551.691} C_VEL
LIN {X 0,Y 477.098,Z 436.822,A -85,B 0,C 180,E1 19550.889,E2 19550.889} C_VEL
LIN {X 0,Y 474.545,Z 511.706,A -85,B 0,C 180,E1 19549.542,E2 19549.542} C_VEL
LIN {X 0,Y 473.593,Z 519.407,A -85,B 0,C 180,E1 19549.495,E2 19549.495} C_VEL
LIN {X 0,Y 468.65,Z 540.015,A -85,B 0,C 180,E1 19549.685,E2 19549.685} C_VEL
LIN {X 0,Y 467.935,Z 546.617,A -85,B 0,C 180,E1 19549.631,E2 19549.631} C_VEL
LIN {X 0,Y 462.335,Z 712.658,A -85,B 0,C 180,E1 19546.639,E2 19546.639} C_VEL
LIN {X 0,Y 460.703,Z 735.99,A -85,B 0,C 180,E1 19546.027,E2 19546.027} C_VEL
LIN {X 0,Y 458.662,Z 758.42,A -85,B 0,C 180,E1 19545.225,E2 19545.225} C_VEL
LIN {X 0,Y 456.241,Z 778.955,A -85,B 0,C 180,E1 19544.269,E2 19544.269} C_VEL
LIN {X 0,Y 453.527,Z 799.315,A -85,B 0,C 180,E1 19543.121,E2 19543.121} C_VEL
LIN {X 0,Y 450.267,Z 820.189,A -85,B 0,C 180,E1 19541.682,E2 19541.682} C_VEL
LIN {X 0,Y 446.934,Z 840.184,A -85,B 0,C 180,E1 19540.045,E2 19540.045} C_VEL
LIN {X 0,Y 443.647,Z 858.279,A -85,B 0,C 180,E1 19538.289,E2 19538.289} C_VEL
LIN {X 0,Y 440.118,Z 876.981,A -85,B 0,C 180,E1 19536.181,E2 19536.181} C_VEL
LIN {X 0,Y 437.039,Z 893.082,A -85,B 0,C 180,E1 19534.06,E2 19534.06} C_VEL
LIN {X 0,Y 433.93,Z 909.329,A -85,B 0,C 180,E1 19531.58,E2 19531.58} C_VEL
LIN {X 0,Y 431.208,Z 924.18,A -85,B 0,C 180,E1 19528.933,E2 19528.933} C_VEL
LIN {X 0,Y 428.889,Z 937.652,A -85,B 0,C 180,E1 19526.12,E2 19526.12} C_VEL
LIN {X 0,Y 427.018,Z 949.814,A -85,B 0,C 180,E1 19523.121,E2 19523.121} C_VEL
LIN {X 0,Y 425.616,Z 961.001,A -85,B 0,C 180,E1 19519.842,E2 19519.842} C_VEL
LIN {X 0,Y 424.773,Z 969.497,A -85,B 0,C 180,E1 19516.798,E2 19516.798} C_VEL
LIN {X 0,Y 424.254,Z 976.417,A -85,B 0,C 180,E1 19513.709,E2 19513.709} C_VEL
LIN {X 0,Y 424.004,Z 981.585,A -85,B 0,C 180,E1 19510.719,E2 19510.719} C_VEL
LIN {X 0,Y 423.917,Z 985.098,A -85,B 0,C 180,E1 19507.825,E2 19507.825} C_VEL
LIN {X 0,Y 423.913,Z 987.233,A -85,B 0,C 180,E1 19504.874,E2 19504.874} C_VEL
LIN {X 0,Y 423.906,Z 987.989,A -85,B 0,C 180,E1 19501.85,E2 19501.85} C_VEL
LIN {X 0,Y 423.914,Z 987.169,A -85,B 0,C 180,E1 19498.892,E2 19498.892} C_VEL
LIN {X 0,Y 423.916,Z 984.849,A -85,B 0,C 180,E1 19495.847,E2 19495.847} C_VEL
LIN {X 0,Y 424.017,Z 981.368,A -85,B 0,C 180,E1 19493.033,E2 19493.033} C_VEL
LIN {X 0,Y 424.3,Z 975.989,A -85,B 0,C 180,E1 19489.984,E2 19489.984} C_VEL
LIN {X 0,Y 424.822,Z 968.828,A -85,B 0,C 180,E1 19486.855,E2 19486.855} C_VEL
LIN {X 0,Y 425.681,Z 960.31,A -85,B 0,C 180,E1 19483.851,E2 19483.851} C_VEL
LIN {X 0,Y 427.119,Z 949.145,A -85,B 0,C 180,E1 19480.601,E2 19480.601} C_VEL
LIN {X 0,Y 429.043,Z 936.817,A -85,B 0,C 180,E1 19477.591,E2 19477.591} C_VEL
LIN {X 0,Y 431.533,Z 922.616,A -85,B 0,C 180,E1 19474.657,E2 19474.657} C_VEL
LIN {X 0,Y 434.399,Z 907.25,A -85,B 0,C 180,E1 19471.965,E2 19471.965} C_VEL
LIN {X 0,Y 437.42,Z 891.344,A -85,B 0,C 180,E1 19469.587,E2 19469.587} C_VEL
LIN {X 0,Y 440.801,Z 874.012,A -85,B 0,C 180,E1 19467.344,E2 19467.344} C_VEL
LIN {X 0,Y 444.089,Z 856.336,A -85,B 0,C 180,E1 19465.399,E2 19465.399} C_VEL
LIN {X 0,Y 447.55,Z 837.05,A -85,B 0,C 180,E1 19463.572,E2 19463.572} C_VEL
LIN {X 0,Y 450.627,Z 818.567,A -85,B 0,C 180,E1 19462.092,E2 19462.092} C_VEL
LIN {X 0,Y 453.909,Z 796.95,A -85,B 0,C 180,E1 19460.637,E2 19460.637} C_VEL
LIN {X 0,Y 456.432,Z 778.023,A -85,B 0,C 180,E1 19459.583,E2 19459.583} C_VEL
LIN {X 0,Y 459.017,Z 754.879,A -85,B 0,C 180,E1 19458.54,E2 19458.54} C_VEL
LIN {X 0,Y 460.95,Z 733.37,A -85,B 0,C 180,E1 19457.795,E2 19457.795} C_VEL
LIN {X 0,Y 462.459,Z 709.889,A -85,B 0,C 180,E1 19457.217,E2 19457.217} C_VEL
LIN {X 0,Y 469.965,Z 497.074,A -85,B 0,C 180,E1 19453.353,E2 19453.353} C_VEL
LIN {X 0,Y 472.055,Z 440.345,A -85,B 0,C 180,E1 19452.291,E2 19452.291} C_VEL
LIN {X 0,Y 461.346,Z 424.747,A -85,B 0,C 180,E1 19450.204,E2 19450.204} C_VEL
LIN {X 0,Y 452.481,Z 412.501,A -85,B 0,C 180,E1 19448.291,E2 19448.291} C_VEL
LIN {X 0,Y 447.554,Z 406.272,A -85,B 0,C 180,E1 19447.145,E2 19447.145} C_VEL
LIN {X 0,Y 444.118,Z 401.776,A -85,B 0,C 180,E1 19446.302,E2 19446.302} C_VEL
LIN {X 0,Y 440.703,Z 397.353,A -85,B 0,C 180,E1 19445.403,E2 19445.403} C_VEL
LIN {X 0,Y 436.625,Z 392.753,A -85,B 0,C 180,E1 19444.302,E2 19444.302} C_VEL
LIN {X 0,Y 435.229,Z 390.623,A -85,B 0,C 180,E1 19443.886,E2 19443.886} C_VEL
LIN {X 0,Y 432.173,Z 387.759,A -85,B 0,C 180,E1 19442.984,E2 19442.984} C_VEL
LIN {X 0,Y 430.316,Z 384.548,A -85,B 0,C 180,E1 19442.357,E2 19442.357} C_VEL
LIN {X 0,Y 427.164,Z 382.276,A -85,B 0,C 180,E1 19441.375,E2 19441.375} C_VEL
LIN {X 0,Y 425.496,Z 379.037,A -85,B 0,C 180,E1 19440.674,E2 19440.674} C_VEL
LIN {X 0,Y 425.325,Z 378.092,A -85,B 0,C 180,E1 19440.068,E2 19440.068} C_VEL
LIN {X 0,Y 425.315,Z 378.064,A -85,B 0,C 180,E1 19436.226,E2 19436.226} C_VEL
LIN {X 0,Y 425.322,Z 378.067,A -85,B 0,C 180,E1 19432.3,E2 19432.3} C_VEL
LIN {X 0,Y 425.319,Z 378.069,A -85,B 0,C 180,E1 19428.474,E2 19428.474} C_VEL
LIN {X 0,Y 425.312,Z 378.068,A -85,B 0,C 180,E1 19424.595,E2 19424.595} C_VEL
LIN {X 0,Y 425.288,Z 378.074,A -85,B 0,C 180,E1 19420.784,E2 19420.784} C_VEL
LIN {X 0,Y 425.272,Z 378.066,A -85,B 0,C 180,E1 19417.028,E2 19417.028} C_VEL
LIN {X 0,Y 425.272,Z 378.062,A -85,B 0,C 180,E1 19413.166,E2 19413.166} C_VEL
LIN {X 0,Y 425.382,Z 378.581,A -85,B 0,C 180,E1 19412.234,E2 19412.234} C_VEL
LIN {X 0,Y 427.091,Z 382.239,A -85,B 0,C 180,E1 19411.116,E2 19411.116} C_VEL
LIN {X 0,Y 429.492,Z 384.816,A -85,B 0,C 180,E1 19410.312,E2 19410.312} C_VEL
LIN {X 0,Y 432.653,Z 388.829,A -85,B 0,C 180,E1 19409.286,E2 19409.286} C_VEL
LIN {X 0,Y 434.061,Z 390.578,A -85,B 0,C 180,E1 19408.86,E2 19408.86} C_VEL
LIN {X 0,Y 439.199,Z 397.361,A -85,B 0,C 180,E1 19407.39,E2 19407.39} C_VEL
LIN {X 0,Y 442.678,Z 402.101,A -85,B 0,C 180,E1 19406.449,E2 19406.449} C_VEL
LIN {X 0,Y 446.857,Z 407.759,A -85,B 0,C 180,E1 19405.405,E2 19405.405} C_VEL
LIN {X 0,Y 455.115,Z 419.555,A -85,B 0,C 180,E1 19403.481,E2 19403.481} C_VEL
LIN {X 0,Y 465.566,Z 435.747,A -85,B 0,C 180,E1 19401.282,E2 19401.282} C_VEL
LIN {X 0,Y 472.182,Z 447.076,A -85,B 0,C 180,E1 19399.991,E2 19399.991} C_VEL
LIN {X 0,Y 465.035,Z 646.209,A -85,B 0,C 180,E1 19396.356,E2 19396.356} C_VEL
LIN {X 0,Y 461.869,Z 738.733,A -85,B 0,C 180,E1 19394.676,E2 19394.676} C_VEL
LIN {X 0,Y 460.063,Z 762.147,A -85,B 0,C 180,E1 19394.061,E2 19394.061} C_VEL
LIN {X 0,Y 457.886,Z 784.867,A -85,B 0,C 180,E1 19393.248,E2 19393.248} C_VEL
LIN {X 0,Y 455.376,Z 805.818,A -85,B 0,C 180,E1 19392.274,E2 19392.274} C_VEL
LIN {X 0,Y 452.411,Z 827.726,A -85,B 0,C 180,E1 19391.028,E2 19391.028} C_VEL
LIN {X 0,Y 449.351,Z 847.624,A -85,B 0,C 180,E1 19389.657,E2 19389.657} C_VEL
LIN {X 0,Y 445.739,Z 869.568,A -85,B 0,C 180,E1 19387.854,E2 19387.854} C_VEL
LIN {X 0,Y 442.525,Z 888.175,A -85,B 0,C 180,E1 19386.052,E2 19386.052} C_VEL
LIN {X 0,Y 439.201,Z 906.464,A -85,B 0,C 180,E1 19383.982,E2 19383.982} C_VEL
LIN {X 0,Y 436.133,Z 923.739,A -85,B 0,C 180,E1 19381.731,E2 19381.731} C_VEL
LIN {X 0,Y 433.215,Z 939.919,A -85,B 0,C 180,E1 19379.26,E2 19379.26} C_VEL
LIN {X 0,Y 430.708,Z 954.925,A -85,B 0,C 180,E1 19376.621,E2 19376.621} C_VEL
LIN {X 0,Y 428.752,Z 967.311,A -85,B 0,C 180,E1 19374.089,E2 19374.089} C_VEL
LIN {X 0,Y 426.928,Z 980.261,A -85,B 0,C 180,E1 19371.001,E2 19371.001} C_VEL
LIN {X 0,Y 425.776,Z 989.504,A -85,B 0,C 180,E1 19368.345,E2 19368.345} C_VEL
LIN {X 0,Y 424.855,Z 998.482,A -85,B 0,C 180,E1 19365.228,E2 19365.228} C_VEL
LIN {X 0,Y 424.345,Z 1005.157,A -85,B 0,C 180,E1 19362.385,E2 19362.385} C_VEL
LIN {X 0,Y 424.052,Z 1010.837,A -85,B 0,C 180,E1 19359.23,E2 19359.23} C_VEL
LIN {X 0,Y 423.949,Z 1014.433,A -85,B 0,C 180,E1 19356.504,E2 19356.504} C_VEL
LIN {X 0,Y 423.888,Z 1016.982,A -85,B 0,C 180,E1 19353.385,E2 19353.385} C_VEL
LIN {X 0,Y 423.887,Z 1017.87,A -85,B 0,C 180,E1 19350.815,E2 19350.815} C_VEL
LIN {X 0,Y 423.911,Z 1017.597,A -85,B 0,C 180,E1 19347.841,E2 19347.841} C_VEL
LIN {X 0,Y 423.915,Z 1015.844,A -85,B 0,C 180,E1 19344.998,E2 19344.998} C_VEL
LIN {X 0,Y 423.994,Z 1012.757,A -85,B 0,C 180,E1 19342.067,E2 19342.067} C_VEL
LIN {X 0,Y 424.178,Z 1007.835,A -85,B 0,C 180,E1 19338.998,E2 19338.998} C_VEL
LIN {X 0,Y 424.573,Z 1001.841,A -85,B 0,C 180,E1 19336.106,E2 19336.106} C_VEL
LIN {X 0,Y 425.277,Z 993.919,A -85,B 0,C 180,E1 19333.113,E2 19333.113} C_VEL
LIN {X 0,Y 426.325,Z 984.947,A -85,B 0,C 180,E1 19330.267,E2 19330.267} C_VEL
LIN {X 0,Y 427.752,Z 974.132,A -85,B 0,C 180,E1 19327.464,E2 19327.464} C_VEL
LIN {X 0,Y 429.676,Z 961.515,A -85,B 0,C 180,E1 19324.654,E2 19324.654} C_VEL
LIN {X 0,Y 431.851,Z 948.174,A -85,B 0,C 180,E1 19322.121,E2 19322.121} C_VEL
LIN {X 0,Y 434.627,Z 932.467,A -85,B 0,C 180,E1 19319.524,E2 19319.524} C_VEL
LIN {X 0,Y 437.528,Z 916.429,A -85,B 0,C 180,E1 19317.242,E2 19317.242} C_VEL
LIN {X 0,Y 440.951,Z 897.666,A -85,B 0,C 180,E1 19314.941,E2 19314.941} C_VEL
LIN {X 0,Y 444.271,Z 879.282,A -85,B 0,C 180,E1 19313,E2 19313} C_VEL
LIN {X 0,Y 447.556,Z 860.153,A -85,B 0,C 180,E1 19311.286,E2 19311.286} C_VEL
LIN {X 0,Y 450.701,Z 840.891,A -85,B 0,C 180,E1 19309.799,E2 19309.799} C_VEL
LIN {X 0,Y 453.734,Z 819.974,A -85,B 0,C 180,E1 19308.456,E2 19308.456} C_VEL
LIN {X 0,Y 456.609,Z 798.217,A -85,B 0,C 180,E1 19307.298,E2 19307.298} C_VEL
LIN {X 0,Y 459.019,Z 776.124,A -85,B 0,C 180,E1 19306.38,E2 19306.38} C_VEL
LIN {X 0,Y 461.105,Z 752.896,A -85,B 0,C 180,E1 19305.641,E2 19305.641} C_VEL
LIN {X 0,Y 462.418,Z 730.824,A -85,B 0,C 180,E1 19305.143,E2 19305.143} C_VEL
LIN {X 0,Y 469.343,Z 521.268,A -85,B 0,C 180,E1 19301.382,E2 19301.382} C_VEL
LIN {X 0,Y 471.862,Z 446.657,A -85,B 0,C 180,E1 19300.003,E2 19300.003} C_VEL
LIN {X 0,Y 461.089,Z 429.933,A -85,B 0,C 180,E1 19298.013,E2 19298.013} C_VEL
LIN {X 0,Y 452.063,Z 416.742,A -85,B 0,C 180,E1 19296.234,E2 19296.234} C_VEL
LIN {X 0,Y 442.367,Z 403.206,A -85,B 0,C 180,E1 19294.171,E2 19294.171} C_VEL
LIN {X 0,Y 438.08,Z 397.498,A -85,B 0,C 180,E1 19293.213,E2 19293.213} C_VEL
LIN {X 0,Y 434.25,Z 392.509,A -85,B 0,C 180,E1 19292.337,E2 19292.337} C_VEL
LIN {X 0,Y 430.201,Z 387.26,A -85,B 0,C 180,E1 19291.373,E2 19291.373} C_VEL
LIN {X 0,Y 428.281,Z 384.233,A -85,B 0,C 180,E1 19290.748,E2 19290.748} C_VEL
LIN {X 0,Y 426.762,Z 381.742,A -85,B 0,C 180,E1 19290.091,E2 19290.091} C_VEL
LIN {X 0,Y 425.275,Z 378.296,A -85,B 0,C 180,E1 19289.181,E2 19289.181} C_VEL
LIN {X 0,Y 425.286,Z 378.062,A -85,B 0,C 180,E1 19285.781,E2 19285.781} C_VEL
LIN {X 0,Y 425.282,Z 378.073,A -85,B 0,C 180,E1 19281.951,E2 19281.951} C_VEL
LIN {X 0,Y 425.254,Z 378.07,A -85,B 0,C 180,E1 19278.222,E2 19278.222} C_VEL
LIN {X 0,Y 425.243,Z 378.066,A -85,B 0,C 180,E1 19274.571,E2 19274.571} C_VEL
LIN {X 0,Y 425.259,Z 378.071,A -85,B 0,C 180,E1 19270.841,E2 19270.841} C_VEL
LIN {X 0,Y 425.3,Z 378.072,A -85,B 0,C 180,E1 19267.157,E2 19267.157} C_VEL
LIN {X 0,Y 425.295,Z 378.069,A -85,B 0,C 180,E1 19263.369,E2 19263.369} C_VEL
LIN {X 0,Y 425.265,Z 378.071,A -85,B 0,C 180,E1 19259.73,E2 19259.73} C_VEL
LIN {X 0,Y 425.259,Z 378.068,A -85,B 0,C 180,E1 19255.955,E2 19255.955} C_VEL
LIN {X 0,Y 425.267,Z 378.061,A -85,B 0,C 180,E1 19252.162,E2 19252.162} C_VEL
LIN {X 0,Y 425.296,Z 378.061,A -85,B 0,C 180,E1 19248.472,E2 19248.472} C_VEL
LIN {X 0,Y 425.323,Z 378.059,A -85,B 0,C 180,E1 19244.734,E2 19244.734} C_VEL
LIN {X 0,Y 425.296,Z 378.063,A -85,B 0,C 180,E1 19240.906,E2 19240.906} C_VEL
LIN {X 0,Y 425.279,Z 378.069,A -85,B 0,C 180,E1 19237.148,E2 19237.148} C_VEL
LIN {X 0,Y 425.276,Z 378.072,A -85,B 0,C 180,E1 19233.291,E2 19233.291} C_VEL
LIN {X 0,Y 425.283,Z 378.071,A -85,B 0,C 180,E1 19229.48,E2 19229.48} C_VEL
LIN {X 0,Y 425.307,Z 378.063,A -85,B 0,C 180,E1 19225.814,E2 19225.814} C_VEL
LIN {X 0,Y 425.325,Z 378.057,A -85,B 0,C 180,E1 19221.945,E2 19221.945} C_VEL
LIN {X 0,Y 425.317,Z 378.061,A -85,B 0,C 180,E1 19218.114,E2 19218.114} C_VEL
LIN {X 0,Y 425.301,Z 378.071,A -85,B 0,C 180,E1 19214.277,E2 19214.277} C_VEL
LIN {X 0,Y 425.292,Z 378.062,A -85,B 0,C 180,E1 19210.449,E2 19210.449} C_VEL
LIN {X 0,Y 425.292,Z 378.07,A -85,B 0,C 180,E1 19206.659,E2 19206.659} C_VEL
LIN {X 0,Y 425.303,Z 378.036,A -85,B 0,C 180,E1 19202.886,E2 19202.886} C_VEL
LIN {X 0,Y 425.341,Z 378.224,A -85,B 0,C 180,E1 19201.53,E2 19201.53} C_VEL
LIN {X 0,Y 425.65,Z 379.544,A -85,B 0,C 180,E1 19201.202,E2 19201.202} C_VEL
LIN {X 0,Y 427.426,Z 382.557,A -85,B 0,C 180,E1 19200.719,E2 19200.719} C_VEL
LIN {X 0,Y 430.135,Z 384.828,A -85,B 0,C 180,E1 19200.082,E2 19200.082} C_VEL
LIN {X 0,Y 432.626,Z 388.628,A -85,B 0,C 180,E1 19199.46,E2 19199.46} C_VEL
LIN {X 0,Y 434.826,Z 390.786,A -85,B 0,C 180,E1 19198.961,E2 19198.961} C_VEL
LIN {X 0,Y 437.873,Z 394.923,A -85,B 0,C 180,E1 19198.255,E2 19198.255} C_VEL
LIN {X 0,Y 439.726,Z 397.134,A -85,B 0,C 180,E1 19197.845,E2 19197.845} C_VEL
LIN {X 0,Y 444.75,Z 403.522,A -85,B 0,C 180,E1 19196.76,E2 19196.76} C_VEL
LIN {X 0,Y 452.104,Z 413.027,A -85,B 0,C 180,E1 19195.239,E2 19195.239} C_VEL
LIN {X 0,Y 463.106,Z 428.039,A -85,B 0,C 180,E1 19193.11,E2 19193.11} C_VEL
LIN {X 0,Y 471.696,Z 440.565,A -85,B 0,C 180,E1 19191.553,E2 19191.553} C_VEL
LIN {X 0,Y 467.935,Z 546.617,A -85,B 0,C 180,E1 19189.631,E2 19189.631} C_VEL
LIN {X 0,Y 467.015,Z 554.315,A -85,B 0,C 180,E1 19189.58,E2 19189.58} C_VEL
LIN {X 0,Y 462.044,Z 574.918,A -85,B 0,C 180,E1 19189.777,E2 19189.777} C_VEL
LIN {X 0,Y 461.294,Z 581.526,A -85,B 0,C 180,E1 19189.727,E2 19189.727} C_VEL
LIN {X 0,Y 456.598,Z 713.269,A -85,B 0,C 180,E1 19187.33,E2 19187.33} C_VEL
LIN {X 0,Y 454.886,Z 736.492,A -85,B 0,C 180,E1 19186.714,E2 19186.714} C_VEL
LIN {X 0,Y 452.787,Z 758.525,A -85,B 0,C 180,E1 19185.92,E2 19185.92} C_VEL
LIN {X 0,Y 450.178,Z 779.7,A -85,B 0,C 180,E1 19184.925,E2 19184.925} C_VEL
LIN {X 0,Y 447.188,Z 800.992,A -85,B 0,C 180,E1 19183.705,E2 19183.705} C_VEL
LIN {X 0,Y 443.861,Z 821.199,A -85,B 0,C 180,E1 19182.286,E2 19182.286} C_VEL
LIN {X 0,Y 440.278,Z 841.491,A -85,B 0,C 180,E1 19180.595,E2 19180.595} C_VEL
LIN {X 0,Y 436.952,Z 858.901,A -85,B 0,C 180,E1 19178.881,E2 19178.881} C_VEL
LIN {X 0,Y 433.139,Z 877.999,A -85,B 0,C 180,E1 19176.69,E2 19176.69} C_VEL
LIN {X 0,Y 429.882,Z 894.098,A -85,B 0,C 180,E1 19174.531,E2 19174.531} C_VEL
LIN {X 0,Y 426.596,Z 910.241,A -85,B 0,C 180,E1 19172.011,E2 19172.011} C_VEL
LIN {X 0,Y 423.718,Z 925.051,A -85,B 0,C 180,E1 19169.32,E2 19169.32} C_VEL
LIN {X 0,Y 421.25,Z 938.434,A -85,B 0,C 180,E1 19166.458,E2 19166.458} C_VEL
LIN {X 0,Y 419.26,Z 950.438,A -85,B 0,C 180,E1 19163.423,E2 19163.423} C_VEL
LIN {X 0,Y 417.835,Z 960.614,A -85,B 0,C 180,E1 19160.353,E2 19160.353} C_VEL
LIN {X 0,Y 416.854,Z 969.444,A -85,B 0,C 180,E1 19157.107,E2 19157.107} C_VEL
LIN {X 0,Y 416.299,Z 976.366,A -85,B 0,C 180,E1 19153.962,E2 19153.962} C_VEL
LIN {X 0,Y 416.016,Z 981.66,A -85,B 0,C 180,E1 19150.831,E2 19150.831} C_VEL
LIN {X 0,Y 415.919,Z 985.063,A -85,B 0,C 180,E1 19147.971,E2 19147.971} C_VEL
LIN {X 0,Y 415.913,Z 987.216,A -85,B 0,C 180,E1 19144.966,E2 19144.966} C_VEL
LIN {X 0,Y 415.907,Z 987.995,A -85,B 0,C 180,E1 19141.885,E2 19141.885} C_VEL
LIN {X 0,Y 415.913,Z 987.177,A -85,B 0,C 180,E1 19138.852,E2 19138.852} C_VEL
LIN {X 0,Y 415.92,Z 984.885,A -85,B 0,C 180,E1 19135.766,E2 19135.766} C_VEL
LIN {X 0,Y 416.032,Z 981.412,A -85,B 0,C 180,E1 19132.895,E2 19132.895} C_VEL
LIN {X 0,Y 416.331,Z 976.067,A -85,B 0,C 180,E1 19129.793,E2 19129.793} C_VEL
LIN {X 0,Y 416.893,Z 968.957,A -85,B 0,C 180,E1 19126.611,E2 19126.611} C_VEL
LIN {X 0,Y 417.922,Z 959.937,A -85,B 0,C 180,E1 19123.335,E2 19123.335} C_VEL
LIN {X 0,Y 419.408,Z 949.627,A -85,B 0,C 180,E1 19120.246,E2 19120.246} C_VEL
LIN {X 0,Y 421.432,Z 937.532,A -85,B 0,C 180,E1 19117.229,E2 19117.229} C_VEL
LIN {X 0,Y 424.028,Z 923.715,A -85,B 0,C 180,E1 19114.303,E2 19114.303} C_VEL
LIN {X 0,Y 426.819,Z 909.487,A -85,B 0,C 180,E1 19111.745,E2 19111.745} C_VEL
LIN {X 0,Y 430.142,Z 893.163,A -85,B 0,C 180,E1 19109.219,E2 19109.219} C_VEL
LIN {X 0,Y 433.535,Z 876.664,A -85,B 0,C 180,E1 19107.023,E2 19107.023} C_VEL
LIN {X 0,Y 437.121,Z 858.585,A -85,B 0,C 180,E1 19104.97,E2 19104.97} C_VEL
LIN {X 0,Y 440.776,Z 839.509,A -85,B 0,C 180,E1 19103.107,E2 19103.107} C_VEL
LIN {X 0,Y 444.153,Z 820.199,A -85,B 0,C 180,E1 19101.527,E2 19101.527} C_VEL
LIN {X 0,Y 447.434,Z 800.08,A -85,B 0,C 180,E1 19100.13,E2 19100.13} C_VEL
LIN {X 0,Y 450.262,Z 779.899,A -85,B 0,C 180,E1 19098.979,E2 19098.979} C_VEL
LIN {X 0,Y 452.894,Z 758.241,A -85,B 0,C 180,E1 19097.968,E2 19097.968} C_VEL
LIN {X 0,Y 454.943,Z 736.689,A -85,B 0,C 180,E1 19097.192,E2 19097.192} C_VEL
LIN {X 0,Y 456.651,Z 712.938,A -85,B 0,C 180,E1 19096.569,E2 19096.569} C_VEL
LIN {X 0,Y 464.622,Z 501.329,A -85,B 0,C 180,E1 19092.678,E2 19092.678} C_VEL
LIN {X 0,Y 466.85,Z 444.381,A -85,B 0,C 180,E1 19091.599,E2 19091.599} C_VEL
LIN {X 0,Y 456.073,Z 428.491,A -85,B 0,C 180,E1 19089.4,E2 19089.4} C_VEL
LIN {X 0,Y 447.957,Z 417.483,A -85,B 0,C 180,E1 19087.568,E2 19087.568} C_VEL
LIN {X 0,Y 444.546,Z 413.022,A -85,B 0,C 180,E1 19086.749,E2 19086.749} C_VEL
LIN {X 0,Y 441.052,Z 408.443,A -85,B 0,C 180,E1 19085.856,E2 19085.856} C_VEL
LIN {X 0,Y 436.989,Z 403.275,A -85,B 0,C 180,E1 19084.758,E2 19084.758} C_VEL
LIN {X 0,Y 433.624,Z 399.137,A -85,B 0,C 180,E1 19083.802,E2 19083.802} C_VEL
LIN {X 0,Y 432.62,Z 397.778,A -85,B 0,C 180,E1 19083.491,E2 19083.491} C_VEL
LIN {X 0,Y 429.414,Z 394.38,A -85,B 0,C 180,E1 19082.506,E2 19082.506} C_VEL
LIN {X 0,Y 427.969,Z 391.956,A -85,B 0,C 180,E1 19082.009,E2 19082.009} C_VEL
LIN {X 0,Y 424.855,Z 389.37,A -85,B 0,C 180,E1 19080.982,E2 19080.982} C_VEL
LIN {X 0,Y 422.743,Z 385.732,A -85,B 0,C 180,E1 19080.136,E2 19080.136} C_VEL
LIN {X 0,Y 419.444,Z 383.496,A -85,B 0,C 180,E1 19078.908,E2 19078.908} C_VEL
LIN {X 0,Y 417.712,Z 380.554,A -85,B 0,C 180,E1 19078.08,E2 19078.08} C_VEL
LIN {X 0,Y 417.395,Z 379.276,A -85,B 0,C 180,E1 19077.529,E2 19077.529} C_VEL
LIN {X 0,Y 417.368,Z 379.048,A -85,B 0,C 180,E1 19073.812,E2 19073.812} C_VEL
LIN {X 0,Y 417.373,Z 379.06,A -85,B 0,C 180,E1 19069.929,E2 19069.929} C_VEL
LIN {X 0,Y 417.385,Z 379.055,A -85,B 0,C 180,E1 19065.983,E2 19065.983} C_VEL
LIN {X 0,Y 417.383,Z 379.059,A -85,B 0,C 180,E1 19062.144,E2 19062.144} C_VEL
LIN {X 0,Y 417.381,Z 379.052,A -85,B 0,C 180,E1 19058.204,E2 19058.204} C_VEL
LIN {X 0,Y 417.365,Z 379.302,A -85,B 0,C 180,E1 19054.903,E2 19054.903} C_VEL
LIN {X 0,Y 417.833,Z 380.943,A -85,B 0,C 180,E1 19054.296,E2 19054.296} C_VEL
LIN {X 0,Y 419.816,Z 383.903,A -85,B 0,C 180,E1 19053.401,E2 19053.401} C_VEL
LIN {X 0,Y 422.396,Z 386.077,A -85,B 0,C 180,E1 19052.396,E2 19052.396} C_VEL
LIN {X 0,Y 426.333,Z 390.961,A -85,B 0,C 180,E1 19050.958,E2 19050.958} C_VEL
LIN {X 0,Y 430.467,Z 396.201,A -85,B 0,C 180,E1 19049.579,E2 19049.579} C_VEL
LIN {X 0,Y 436.584,Z 404.423,A -85,B 0,C 180,E1 19047.751,E2 19047.751} C_VEL
LIN {X 0,Y 443.176,Z 413.478,A -85,B 0,C 180,E1 19045.978,E2 19045.978} C_VEL
LIN {X 0,Y 451.935,Z 426.321,A -85,B 0,C 180,E1 19043.864,E2 19043.864} C_VEL
LIN {X 0,Y 461.7,Z 441.639,A -85,B 0,C 180,E1 19041.751,E2 19041.751} C_VEL
LIN {X 0,Y 466.969,Z 450.752,A -85,B 0,C 180,E1 19040.684,E2 19040.684} C_VEL
LIN {X 0,Y 459.393,Z 649.158,A -85,B 0,C 180,E1 19037.022,E2 19037.022} C_VEL
LIN {X 0,Y 456.152,Z 738.308,A -85,B 0,C 180,E1 19035.385,E2 19035.385} C_VEL
LIN {X 0,Y 454.263,Z 761.689,A -85,B 0,C 180,E1 19034.768,E2 19034.768} C_VEL
LIN {X 0,Y 451.977,Z 784.296,A -85,B 0,C 180,E1 19033.957,E2 19033.957} C_VEL
LIN {X 0,Y 449.267,Z 805.82,A -85,B 0,C 180,E1 19032.949,E2 19032.949} C_VEL
LIN {X 0,Y 446.062,Z 828.227,A -85,B 0,C 180,E1 19031.656,E2 19031.656} C_VEL
LIN {X 0,Y 442.977,Z 847.289,A -85,B 0,C 180,E1 19030.326,E2 19030.326} C_VEL
LIN {X 0,Y 439.162,Z 869.161,A -85,B 0,C 180,E1 19028.513,E2 19028.513} C_VEL
LIN {X 0,Y 435.794,Z 887.618,A -85,B 0,C 180,E1 19026.707,E2 19026.707} C_VEL
LIN {X 0,Y 432.19,Z 906.401,A -85,B 0,C 180,E1 19024.555,E2 19024.555} C_VEL
LIN {X 0,Y 428.923,Z 923.676,A -85,B 0,C 180,E1 19022.267,E2 19022.267} C_VEL
LIN {X 0,Y 425.937,Z 939.279,A -85,B 0,C 180,E1 19019.848,E2 19019.848} C_VEL
LIN {X 0,Y 423.216,Z 954.521,A -85,B 0,C 180,E1 19017.131,E2 19017.131} C_VEL
LIN {X 0,Y 421.109,Z 966.917,A -85,B 0,C 180,E1 19014.555,E2 19014.555} C_VEL
LIN {X 0,Y 419.222,Z 979.399,A -85,B 0,C 180,E1 19011.541,E2 19011.541} C_VEL
LIN {X 0,Y 417.987,Z 988.873,A -85,B 0,C 180,E1 19008.844,E2 19008.844} C_VEL
LIN {X 0,Y 417.037,Z 997.628,A -85,B 0,C 180,E1 19005.865,E2 19005.865} C_VEL
LIN {X 0,Y 416.453,Z 1004.248,A -85,B 0,C 180,E1 19003.047,E2 19003.047} C_VEL
LIN {X 0,Y 416.074,Z 1010.217,A -85,B 0,C 180,E1 18999.828,E2 18999.828} C_VEL
LIN {X 0,Y 415.939,Z 1013.954,A -85,B 0,C 180,E1 18997.046,E2 18997.046} C_VEL
LIN {X 0,Y 415.91,Z 1016.71,A -85,B 0,C 180,E1 18994.002,E2 18994.002} C_VEL
LIN {X 0,Y 415.897,Z 1017.825,A -85,B 0,C 180,E1 18991.106,E2 18991.106} C_VEL
LIN {X 0,Y 415.906,Z 1017.735,A -85,B 0,C 180,E1 18988.351,E2 18988.351} C_VEL
LIN {X 0,Y 415.911,Z 1016.071,A -85,B 0,C 180,E1 18985.178,E2 18985.178} C_VEL
LIN {X 0,Y 415.95,Z 1013.484,A -85,B 0,C 180,E1 18982.546,E2 18982.546} C_VEL
LIN {X 0,Y 416.139,Z 1009.107,A -85,B 0,C 180,E1 18979.483,E2 18979.483} C_VEL
LIN {X 0,Y 416.52,Z 1003.356,A -85,B 0,C 180,E1 18976.54,E2 18976.54} C_VEL
LIN {X 0,Y 417.256,Z 995.369,A -85,B 0,C 180,E1 18973.294,E2 18973.294} C_VEL
LIN {X 0,Y 418.213,Z 987.045,A -85,B 0,C 180,E1 18970.596,E2 18970.596} C_VEL
LIN {X 0,Y 419.797,Z 975.563,A -85,B 0,C 180,E1 18967.457,E2 18967.457} C_VEL
LIN {X 0,Y 421.657,Z 963.833,A -85,B 0,C 180,E1 18964.739,E2 18964.739} C_VEL
LIN {X 0,Y 424.159,Z 949.402,A -85,B 0,C 180,E1 18961.877,E2 18961.877} C_VEL
LIN {X 0,Y 426.985,Z 934.431,A -85,B 0,C 180,E1 18959.31,E2 18959.31} C_VEL
LIN {X 0,Y 430.123,Z 917.94,A -85,B 0,C 180,E1 18956.894,E2 18956.894} C_VEL
LIN {X 0,Y 433.593,Z 900.215,A -85,B 0,C 180,E1 18954.64,E2 18954.64} C_VEL
LIN {X 0,Y 436.989,Z 882.216,A -85,B 0,C 180,E1 18952.682,E2 18952.682} C_VEL
LIN {X 0,Y 440.828,Z 861.383,A -85,B 0,C 180,E1 18950.749,E2 18950.749} C_VEL
LIN {X 0,Y 443.95,Z 843.177,A -85,B 0,C 180,E1 18949.314,E2 18949.314} C_VEL
LIN {X 0,Y 447.45,Z 820.62,A -85,B 0,C 180,E1 18947.825,E2 18947.825} C_VEL
LIN {X 0,Y 450.46,Z 799.048,A -85,B 0,C 180,E1 18946.66,E2 18946.66} C_VEL
LIN {X 0,Y 453.015,Z 776.947,A -85,B 0,C 180,E1 18945.724,E2 18945.724} C_VEL
LIN {X 0,Y 455.201,Z 754.269,A -85,B 0,C 180,E1 18944.983,E2 18944.983} C_VEL
LIN {X 0,Y 456.645,Z 731.446,A -85,B 0,C 180,E1 18944.457,E2 18944.457} C_VEL
LIN {X 0,Y 464.007,Z 520.867,A -85,B 0,C 180,E1 18940.64,E2 18940.64} C_VEL
LIN {X 0,Y 466.549,Z 450.462,A -85,B 0,C 180,E1 18939.331,E2 18939.331} C_VEL
LIN {X 0,Y 454.24,Z 431.313,A -85,B 0,C 180,E1 18936.971,E2 18936.971} C_VEL
LIN {X 0,Y 441.862,Z 413.539,A -85,B 0,C 180,E1 18934.372,E2 18934.372} C_VEL
LIN {X 0,Y 434.309,Z 403.411,A -85,B 0,C 180,E1 18932.674,E2 18932.674} C_VEL
LIN {X 0,Y 430.747,Z 398.746,A -85,B 0,C 180,E1 18931.836,E2 18931.836} C_VEL
LIN {X 0,Y 426.912,Z 393.71,A -85,B 0,C 180,E1 18930.897,E2 18930.897} C_VEL
LIN {X 0,Y 423.057,Z 388.728,A -85,B 0,C 180,E1 18929.912,E2 18929.912} C_VEL
LIN {X 0,Y 420.171,Z 384.441,A -85,B 0,C 180,E1 18929.041,E2 18929.041} C_VEL
LIN {X 0,Y 417.78,Z 380.805,A -85,B 0,C 180,E1 18927.974,E2 18927.974} C_VEL
LIN {X 0,Y 417.355,Z 379.26,A -85,B 0,C 180,E1 18927.54,E2 18927.54} C_VEL
LIN {X 0,Y 417.351,Z 379.05,A -85,B 0,C 180,E1 18923.786,E2 18923.786} C_VEL
LIN {X 0,Y 417.331,Z 379.055,A -85,B 0,C 180,E1 18920.035,E2 18920.035} C_VEL
LIN {X 0,Y 417.312,Z 379.066,A -85,B 0,C 180,E1 18916.279,E2 18916.279} C_VEL
LIN {X 0,Y 417.309,Z 379.06,A -85,B 0,C 180,E1 18912.452,E2 18912.452} C_VEL
LIN {X 0,Y 417.313,Z 379.052,A -85,B 0,C 180,E1 18908.542,E2 18908.542} C_VEL
LIN {X 0,Y 417.344,Z 379.052,A -85,B 0,C 180,E1 18904.947,E2 18904.947} C_VEL
LIN {X 0,Y 417.371,Z 379.054,A -85,B 0,C 180,E1 18901.098,E2 18901.098} C_VEL
LIN {X 0,Y 417.357,Z 379.061,A -85,B 0,C 180,E1 18897.253,E2 18897.253} C_VEL
LIN {X 0,Y 417.331,Z 379.065,A -85,B 0,C 180,E1 18893.534,E2 18893.534} C_VEL
LIN {X 0,Y 417.326,Z 379.063,A -85,B 0,C 180,E1 18889.787,E2 18889.787} C_VEL
LIN {X 0,Y 417.328,Z 379.057,A -85,B 0,C 180,E1 18885.854,E2 18885.854} C_VEL
LIN {X 0,Y 417.352,Z 379.049,A -85,B 0,C 180,E1 18882.142,E2 18882.142} C_VEL
LIN {X 0,Y 417.383,Z 379.045,A -85,B 0,C 180,E1 18878.335,E2 18878.335} C_VEL
LIN {X 0,Y 417.376,Z 379.048,A -85,B 0,C 180,E1 18874.455,E2 18874.455} C_VEL
LIN {X 0,Y 417.365,Z 379.052,A -85,B 0,C 180,E1 18870.586,E2 18870.586} C_VEL
LIN {X 0,Y 417.344,Z 379.061,A -85,B 0,C 180,E1 18866.89,E2 18866.89} C_VEL
LIN {X 0,Y 417.343,Z 379.062,A -85,B 0,C 180,E1 18863.033,E2 18863.033} C_VEL
LIN {X 0,Y 417.349,Z 379.05,A -85,B 0,C 180,E1 18859.153,E2 18859.153} C_VEL
LIN {X 0,Y 417.365,Z 379.05,A -85,B 0,C 180,E1 18855.349,E2 18855.349} C_VEL
LIN {X 0,Y 417.385,Z 379.056,A -85,B 0,C 180,E1 18851.426,E2 18851.426} C_VEL
LIN {X 0,Y 417.38,Z 379.048,A -85,B 0,C 180,E1 18847.539,E2 18847.539} C_VEL
LIN {X 0,Y 417.379,Z 379.041,A -85,B 0,C 180,E1 18843.592,E2 18843.592} C_VEL
LIN {X 0,Y 417.448,Z 379.492,A -85,B 0,C 180,E1 18843.175,E2 18843.175} C_VEL
LIN {X 0,Y 418.205,Z 381.741,A -85,B 0,C 180,E1 18842.756,E2 18842.756} C_VEL
LIN {X 0,Y 420.463,Z 384.427,A -85,B 0,C 180,E1 18842.159,E2 18842.159} C_VEL
LIN {X 0,Y 422.284,Z 385.831,A -85,B 0,C 180,E1 18841.714,E2 18841.714} C_VEL
LIN {X 0,Y 424.671,Z 389.566,A -85,B 0,C 180,E1 18841.081,E2 18841.081} C_VEL
LIN {X 0,Y 427.264,Z 392.046,A -85,B 0,C 180,E1 18840.451,E2 18840.451} C_VEL
LIN {X 0,Y 430.399,Z 396.225,A -85,B 0,C 180,E1 18839.675,E2 18839.675} C_VEL
LIN {X 0,Y 432.048,Z 398.139,A -85,B 0,C 180,E1 18839.286,E2 18839.286} C_VEL
LIN {X 0,Y 437.09,Z 404.651,A -85,B 0,C 180,E1 18838.119,E2 18838.119} C_VEL
LIN {X 0,Y 441.893,Z 410.722,A -85,B 0,C 180,E1 18837.066,E2 18837.066} C_VEL
LIN {X 0,Y 449.352,Z 420.515,A -85,B 0,C 180,E1 18835.502,E2 18835.502} C_VEL
LIN {X 0,Y 459.375,Z 434.28,A -85,B 0,C 180,E1 18833.525,E2 18833.525} C_VEL
LIN {X 0,Y 466.353,Z 444.509,A -85,B 0,C 180,E1 18832.229,E2 18832.229} C_VEL
LIN {X 0,Y 461.294,Z 581.526,A -85,B 0,C 180,E1 18829.727,E2 18829.727} C_VEL
LIN {X 0,Y 460.338,Z 589.224,A -85,B 0,C 180,E1 18829.679,E2 18829.679} C_VEL
LIN {X 0,Y 455.335,Z 609.813,A -85,B 0,C 180,E1 18829.881,E2 18829.881} C_VEL
LIN {X 0,Y 454.578,Z 616.417,A -85,B 0,C 180,E1 18829.83,E2 18829.83} C_VEL
LIN {X 0,Y 450.896,Z 714.083,A -85,B 0,C 180,E1 18828.031,E2 18828.031} C_VEL
LIN {X 0,Y 449.108,Z 737.144,A -85,B 0,C 180,E1 18827.411,E2 18827.411} C_VEL
LIN {X 0,Y 446.898,Z 759.329,A -85,B 0,C 180,E1 18826.603,E2 18826.603} C_VEL
LIN {X 0,Y 444.175,Z 780.443,A -85,B 0,C 180,E1 18825.6,E2 18825.6} C_VEL
LIN {X 0,Y 441.045,Z 801.661,A -85,B 0,C 180,E1 18824.369,E2 18824.369} C_VEL
LIN {X 0,Y 437.569,Z 821.845,A -85,B 0,C 180,E1 18822.936,E2 18822.936} C_VEL
LIN {X 0,Y 433.795,Z 842.103,A -85,B 0,C 180,E1 18821.226,E2 18821.226} C_VEL
LIN {X 0,Y 430.184,Z 860.125,A -85,B 0,C 180,E1 18819.427,E2 18819.427} C_VEL
LIN {X 0,Y 426.182,Z 879.091,A -85,B 0,C 180,E1 18817.206,E2 18817.206} C_VEL
LIN {X 0,Y 422.569,Z 896.071,A -85,B 0,C 180,E1 18814.882,E2 18814.882} C_VEL
LIN {X 0,Y 419.288,Z 911.158,A -85,B 0,C 180,E1 18812.456,E2 18812.456} C_VEL
LIN {X 0,Y 416.246,Z 925.909,A -85,B 0,C 180,E1 18809.721,E2 18809.721} C_VEL
LIN {X 0,Y 413.6,Z 939.34,A -85,B 0,C 180,E1 18806.776,E2 18806.776} C_VEL
LIN {X 0,Y 411.47,Z 951.358,A -85,B 0,C 180,E1 18803.651,E2 18803.651} C_VEL
LIN {X 0,Y 409.992,Z 961.261,A -85,B 0,C 180,E1 18800.592,E2 18800.592} C_VEL
LIN {X 0,Y 408.963,Z 969.604,A -85,B 0,C 180,E1 18797.428,E2 18797.428} C_VEL
LIN {X 0,Y 408.346,Z 976.386,A -85,B 0,C 180,E1 18794.216,E2 18794.216} C_VEL
LIN {X 0,Y 408.04,Z 981.586,A -85,B 0,C 180,E1 18791.06,E2 18791.06} C_VEL
LIN {X 0,Y 407.925,Z 985.026,A -85,B 0,C 180,E1 18788.122,E2 18788.122} C_VEL
LIN {X 0,Y 407.913,Z 987.267,A -85,B 0,C 180,E1 18784.906,E2 18784.906} C_VEL
LIN {X 0,Y 407.905,Z 987.977,A -85,B 0,C 180,E1 18781.762,E2 18781.762} C_VEL
LIN {X 0,Y 407.91,Z 987.131,A -85,B 0,C 180,E1 18778.688,E2 18778.688} C_VEL
LIN {X 0,Y 407.935,Z 984.748,A -85,B 0,C 180,E1 18775.512,E2 18775.512} C_VEL
LIN {X 0,Y 408.069,Z 981.189,A -85,B 0,C 180,E1 18772.55,E2 18772.55} C_VEL
LIN {X 0,Y 408.417,Z 975.397,A -85,B 0,C 180,E1 18769.155,E2 18769.155} C_VEL
LIN {X 0,Y 409.076,Z 968.545,A -85,B 0,C 180,E1 18766.037,E2 18766.037} C_VEL
LIN {X 0,Y 410.217,Z 959.722,A -85,B 0,C 180,E1 18762.803,E2 18762.803} C_VEL
LIN {X 0,Y 411.782,Z 949.773,A -85,B 0,C 180,E1 18759.782,E2 18759.782} C_VEL
LIN {X 0,Y 413.881,Z 938.046,A -85,B 0,C 180,E1 18756.808,E2 18756.808} C_VEL
LIN {X 0,Y 416.461,Z 925.224,A -85,B 0,C 180,E1 18754.015,E2 18754.015} C_VEL
LIN {X 0,Y 419.396,Z 911.062,A -85,B 0,C 180,E1 18751.403,E2 18751.403} C_VEL
LIN {X 0,Y 422.883,Z 894.984,A -85,B 0,C 180,E1 18748.839,E2 18748.839} C_VEL
LIN {X 0,Y 426.312,Z 879.083,A -85,B 0,C 180,E1 18746.668,E2 18746.668} C_VEL
LIN {X 0,Y 430.361,Z 859.907,A -85,B 0,C 180,E1 18744.428,E2 18744.428} C_VEL
LIN {X 0,Y 434.004,Z 841.869,A -85,B 0,C 180,E1 18742.628,E2 18742.628} C_VEL
LIN {X 0,Y 437.729,Z 821.848,A -85,B 0,C 180,E1 18740.946,E2 18740.946} C_VEL
LIN {X 0,Y 441.256,Z 801.402,A -85,B 0,C 180,E1 18739.497,E2 18739.497} C_VEL
LIN {X 0,Y 444.238,Z 781.169,A -85,B 0,C 180,E1 18738.324,E2 18738.324} C_VEL
LIN {X 0,Y 446.896,Z 760.746,A -85,B 0,C 180,E1 18737.346,E2 18737.346} C_VEL
LIN {X 0,Y 449.145,Z 738.382,A -85,B 0,C 180,E1 18736.52,E2 18736.52} C_VEL
LIN {X 0,Y 450.926,Z 715.776,A -85,B 0,C 180,E1 18735.9,E2 18735.9} C_VEL
LIN {X 0,Y 454.446,Z 626.873,A -85,B 0,C 180,E1 18734.242,E2 18734.242} C_VEL
LIN {X 0,Y 461.806,Z 448.443,A -85,B 0,C 180,E1 18730.905,E2 18730.905} C_VEL
LIN {X 0,Y 451.942,Z 433.93,A -85,B 0,C 180,E1 18728.813,E2 18728.813} C_VEL
LIN {X 0,Y 442.818,Z 421.189,A -85,B 0,C 180,E1 18726.65,E2 18726.65} C_VEL
LIN {X 0,Y 437.795,Z 414.823,A -85,B 0,C 180,E1 18725.344,E2 18725.344} C_VEL
LIN {X 0,Y 434.201,Z 410.181,A -85,B 0,C 180,E1 18724.347,E2 18724.347} C_VEL
LIN {X 0,Y 430.72,Z 405.556,A -85,B 0,C 180,E1 18723.298,E2 18723.298} C_VEL
LIN {X 0,Y 426.86,Z 401.265,A -85,B 0,C 180,E1 18722.081,E2 18722.081} C_VEL
LIN {X 0,Y 425.512,Z 399.248,A -85,B 0,C 180,E1 18721.616,E2 18721.616} C_VEL
LIN {X 0,Y 422.288,Z 396.067,A -85,B 0,C 180,E1 18720.475,E2 18720.475} C_VEL
LIN {X 0,Y 420.635,Z 393.216,A -85,B 0,C 180,E1 18719.796,E2 18719.796} C_VEL
LIN {X 0,Y 417.447,Z 390.827,A -85,B 0,C 180,E1 18718.559,E2 18718.559} C_VEL
LIN {X 0,Y 415.578,Z 387.531,A -85,B 0,C 180,E1 18717.622,E2 18717.622} C_VEL
LIN {X 0,Y 414.468,Z 386.53,A -85,B 0,C 180,E1 18717.097,E2 18717.097} C_VEL
LIN {X 0,Y 411.153,Z 384.1,A -85,B 0,C 180,E1 18715.398,E2 18715.398} C_VEL
LIN {X 0,Y 409.572,Z 380.798,A -85,B 0,C 180,E1 18714.116,E2 18714.116} C_VEL
LIN {X 0,Y 409.442,Z 380.059,A -85,B 0,C 180,E1 18712.846,E2 18712.846} C_VEL
LIN {X 0,Y 409.424,Z 380.047,A -85,B 0,C 180,E1 18708.877,E2 18708.877} C_VEL
LIN {X 0,Y 409.412,Z 380.05,A -85,B 0,C 180,E1 18704.997,E2 18704.997} C_VEL
LIN {X 0,Y 409.405,Z 380.051,A -85,B 0,C 180,E1 18701.046,E2 18701.046} C_VEL
LIN {X 0,Y 409.46,Z 380.38,A -85,B 0,C 180,E1 18698.664,E2 18698.664} C_VEL
LIN {X 0,Y 409.789,Z 381.564,A -85,B 0,C 180,E1 18697.976,E2 18697.976} C_VEL
LIN {X 0,Y 411.535,Z 384.56,A -85,B 0,C 180,E1 18696.822,E2 18696.822} C_VEL
LIN {X 0,Y 415.415,Z 387.401,A -85,B 0,C 180,E1 18694.862,E2 18694.862} C_VEL
LIN {X 0,Y 417.544,Z 390.968,A -85,B 0,C 180,E1 18693.858,E2 18693.858} C_VEL
LIN {X 0,Y 420.468,Z 393.624,A -85,B 0,C 180,E1 18692.681,E2 18692.681} C_VEL
LIN {X 0,Y 424.387,Z 398.5,A -85,B 0,C 180,E1 18691.205,E2 18691.205} C_VEL
LIN {X 0,Y 428.103,Z 403.389,A -85,B 0,C 180,E1 18689.936,E2 18689.936} C_VEL
LIN {X 0,Y 434.29,Z 411.91,A -85,B 0,C 180,E1 18688.027,E2 18688.027} C_VEL
LIN {X 0,Y 440.888,Z 421.247,A -85,B 0,C 180,E1 18686.208,E2 18686.208} C_VEL
LIN {X 0,Y 448.688,Z 432.894,A -85,B 0,C 180,E1 18684.279,E2 18684.279} C_VEL
LIN {X 0,Y 457.987,Z 447.741,A -85,B 0,C 180,E1 18682.204,E2 18682.204} C_VEL
LIN {X 0,Y 461.84,Z 454.554,A -85,B 0,C 180,E1 18681.392,E2 18681.392} C_VEL
LIN {X 0,Y 453.879,Z 650.929,A -85,B 0,C 180,E1 18677.729,E2 18677.729} C_VEL
LIN {X 0,Y 450.504,Z 738.035,A -85,B 0,C 180,E1 18676.109,E2 18676.109} C_VEL
LIN {X 0,Y 448.515,Z 761.549,A -85,B 0,C 180,E1 18675.484,E2 18675.484} C_VEL
LIN {X 0,Y 446.053,Z 784.551,A -85,B 0,C 180,E1 18674.65,E2 18674.65} C_VEL
LIN {X 0,Y 443.257,Z 805.656,A -85,B 0,C 180,E1 18673.653,E2 18673.653} C_VEL
LIN {X 0,Y 439.769,Z 828.734,A -85,B 0,C 180,E1 18672.301,E2 18672.301} C_VEL
LIN {X 0,Y 436.485,Z 848.05,A -85,B 0,C 180,E1 18670.934,E2 18670.934} C_VEL
LIN {X 0,Y 432.536,Z 869.394,A -85,B 0,C 180,E1 18669.133,E2 18669.133} C_VEL
LIN {X 0,Y 428.86,Z 888.496,A -85,B 0,C 180,E1 18667.233,E2 18667.233} C_VEL
LIN {X 0,Y 425.276,Z 906.11,A -85,B 0,C 180,E1 18665.174,E2 18665.174} C_VEL
LIN {X 0,Y 421.829,Z 923.234,A -85,B 0,C 180,E1 18662.878,E2 18662.878} C_VEL
LIN {X 0,Y 418.67,Z 938.857,A -85,B 0,C 180,E1 18660.421,E2 18660.421} C_VEL
LIN {X 0,Y 415.753,Z 954.116,A -85,B 0,C 180,E1 18657.659,E2 18657.659} C_VEL
LIN {X 0,Y 413.501,Z 966.529,A -85,B 0,C 180,E1 18655.038,E2 18655.038} C_VEL
LIN {X 0,Y 411.484,Z 978.986,A -85,B 0,C 180,E1 18651.979,E2 18651.979} C_VEL
LIN {X 0,Y 410.147,Z 988.51,A -85,B 0,C 180,E1 18649.218,E2 18649.218} C_VEL
LIN {X 0,Y 409.049,Z 998.079,A -85,B 0,C 180,E1 18645.892,E2 18645.892} C_VEL
LIN {X 0,Y 408.456,Z 1004.79,A -85,B 0,C 180,E1 18643.019,E2 18643.019} C_VEL
LIN {X 0,Y 408.082,Z 1010.424,A -85,B 0,C 180,E1 18639.88,E2 18639.88} C_VEL
LIN {X 0,Y 407.94,Z 1013.954,A -85,B 0,C 180,E1 18637.185,E2 18637.185} C_VEL
LIN {X 0,Y 407.91,Z 1016.709,A -85,B 0,C 180,E1 18634.08,E2 18634.08} C_VEL
LIN {X 0,Y 407.898,Z 1017.825,A -85,B 0,C 180,E1 18631.128,E2 18631.128} C_VEL
LIN {X 0,Y 407.906,Z 1017.735,A -85,B 0,C 180,E1 18628.319,E2 18628.319} C_VEL
LIN {X 0,Y 407.913,Z 1016.071,A -85,B 0,C 180,E1 18625.083,E2 18625.083} C_VEL
LIN {X 0,Y 407.961,Z 1013.484,A -85,B 0,C 180,E1 18622.399,E2 18622.399} C_VEL
LIN {X 0,Y 408.176,Z 1008.962,A -85,B 0,C 180,E1 18619.194,E2 18619.194} C_VEL
LIN {X 0,Y 408.548,Z 1003.568,A -85,B 0,C 180,E1 18616.417,E2 18616.417} C_VEL
LIN {X 0,Y 409.278,Z 995.891,A -85,B 0,C 180,E1 18613.251,E2 18613.251} C_VEL
LIN {X 0,Y 410.326,Z 987.197,A -85,B 0,C 180,E1 18610.355,E2 18610.355} C_VEL
LIN {X 0,Y 411.939,Z 976.269,A -85,B 0,C 180,E1 18607.269,E2 18607.269} C_VEL
LIN {X 0,Y 413.856,Z 964.798,A -85,B 0,C 180,E1 18604.536,E2 18604.536} C_VEL
LIN {X 0,Y 416.475,Z 950.63,A -85,B 0,C 180,E1 18601.624,E2 18601.624} C_VEL
LIN {X 0,Y 419.24,Z 936.652,A -85,B 0,C 180,E1 18599.156,E2 18599.156} C_VEL
LIN {X 0,Y 422.696,Z 919.639,A -85,B 0,C 180,E1 18596.561,E2 18596.561} C_VEL
LIN {X 0,Y 426.197,Z 902.8,A -85,B 0,C 180,E1 18594.346,E2 18594.346} C_VEL
LIN {X 0,Y 429.912,Z 884.188,A -85,B 0,C 180,E1 18592.254,E2 18592.254} C_VEL
LIN {X 0,Y 433.696,Z 865.051,A -85,B 0,C 180,E1 18590.405,E2 18590.405} C_VEL
LIN {X 0,Y 437.303,Z 845.045,A -85,B 0,C 180,E1 18588.783,E2 18588.783} C_VEL
LIN {X 0,Y 440.732,Z 824.695,A -85,B 0,C 180,E1 18587.383,E2 18587.383} C_VEL
LIN {X 0,Y 443.71,Z 804.352,A -85,B 0,C 180,E1 18586.235,E2 18586.235} C_VEL
LIN {X 0,Y 446.631,Z 781.629,A -85,B 0,C 180,E1 18585.197,E2 18585.197} C_VEL
LIN {X 0,Y 448.864,Z 759.955,A -85,B 0,C 180,E1 18584.441,E2 18584.441} C_VEL
LIN {X 0,Y 450.775,Z 734.845,A -85,B 0,C 180,E1 18583.812,E2 18583.812} C_VEL
LIN {X 0,Y 458.532,Z 526.024,A -85,B 0,C 180,E1 18579.983,E2 18579.983} C_VEL
LIN {X 0,Y 461.219,Z 454.187,A -85,B 0,C 180,E1 18578.633,E2 18578.633} C_VEL
LIN {X 0,Y 449.11,Z 435.383,A -85,B 0,C 180,E1 18576.233,E2 18576.233} C_VEL
LIN {X 0,Y 436.55,Z 417.234,A -85,B 0,C 180,E1 18573.502,E2 18573.502} C_VEL
LIN {X 0,Y 427.675,Z 405.454,A -85,B 0,C 180,E1 18571.422,E2 18571.422} C_VEL
LIN {X 0,Y 420.553,Z 395.976,A -85,B 0,C 180,E1 18569.598,E2 18569.598} C_VEL
LIN {X 0,Y 416.285,Z 390.537,A -85,B 0,C 180,E1 18568.435,E2 18568.435} C_VEL
LIN {X 0,Y 413.088,Z 386.505,A -85,B 0,C 180,E1 18567.535,E2 18567.535} C_VEL
LIN {X 0,Y 411.421,Z 384.484,A -85,B 0,C 180,E1 18567.029,E2 18567.029} C_VEL
LIN {X 0,Y 409.61,Z 381.111,A -85,B 0,C 180,E1 18566.064,E2 18566.064} C_VEL
LIN {X 0,Y 409.422,Z 380.185,A -85,B 0,C 180,E1 18565.706,E2 18565.706} C_VEL
LIN {X 0,Y 409.421,Z 380.051,A -85,B 0,C 180,E1 18561.789,E2 18561.789} C_VEL
LIN {X 0,Y 409.397,Z 380.042,A -85,B 0,C 180,E1 18557.922,E2 18557.922} C_VEL
LIN {X 0,Y 409.377,Z 380.044,A -85,B 0,C 180,E1 18554.136,E2 18554.136} C_VEL
LIN {X 0,Y 409.372,Z 380.054,A -85,B 0,C 180,E1 18550.27,E2 18550.27} C_VEL
LIN {X 0,Y 409.375,Z 380.049,A -85,B 0,C 180,E1 18546.309,E2 18546.309} C_VEL
LIN {X 0,Y 409.378,Z 380.041,A -85,B 0,C 180,E1 18542.379,E2 18542.379} C_VEL
LIN {X 0,Y 409.397,Z 380.04,A -85,B 0,C 180,E1 18538.6,E2 18538.6} C_VEL
LIN {X 0,Y 409.424,Z 380.039,A -85,B 0,C 180,E1 18534.815,E2 18534.815} C_VEL
LIN {X 0,Y 409.427,Z 380.041,A -85,B 0,C 180,E1 18531.008,E2 18531.008} C_VEL
LIN {X 0,Y 409.41,Z 380.049,A -85,B 0,C 180,E1 18527.159,E2 18527.159} C_VEL
LIN {X 0,Y 409.395,Z 380.052,A -85,B 0,C 180,E1 18523.396,E2 18523.396} C_VEL
LIN {X 0,Y 409.396,Z 380.051,A -85,B 0,C 180,E1 18519.558,E2 18519.558} C_VEL
LIN {X 0,Y 409.404,Z 380.045,A -85,B 0,C 180,E1 18515.776,E2 18515.776} C_VEL
LIN {X 0,Y 409.434,Z 380.035,A -85,B 0,C 180,E1 18512.038,E2 18512.038} C_VEL
LIN {X 0,Y 409.443,Z 380.035,A -85,B 0,C 180,E1 18508.165,E2 18508.165} C_VEL
LIN {X 0,Y 409.434,Z 380.039,A -85,B 0,C 180,E1 18504.292,E2 18504.292} C_VEL
LIN {X 0,Y 409.423,Z 380.049,A -85,B 0,C 180,E1 18500.402,E2 18500.402} C_VEL
LIN {X 0,Y 409.411,Z 380.043,A -85,B 0,C 180,E1 18496.665,E2 18496.665} C_VEL
LIN {X 0,Y 409.409,Z 380.038,A -85,B 0,C 180,E1 18492.752,E2 18492.752} C_VEL
LIN {X 0,Y 409.417,Z 380.051,A -85,B 0,C 180,E1 18488.868,E2 18488.868} C_VEL
LIN {X 0,Y 409.454,Z 380.177,A -85,B 0,C 180,E1 18485.184,E2 18485.184} C_VEL
LIN {X 0,Y 409.734,Z 381.454,A -85,B 0,C 180,E1 18484.815,E2 18484.815} C_VEL
LIN {X 0,Y 411.521,Z 384.495,A -85,B 0,C 180,E1 18484.238,E2 18484.238} C_VEL
LIN {X 0,Y 414.455,Z 386.882,A -85,B 0,C 180,E1 18483.447,E2 18483.447} C_VEL
LIN {X 0,Y 416.803,Z 390.592,A -85,B 0,C 180,E1 18482.774,E2 18482.774} C_VEL
LIN {X 0,Y 419.482,Z 393.113,A -85,B 0,C 180,E1 18482.087,E2 18482.087} C_VEL
LIN {X 0,Y 422.465,Z 397.152,A -85,B 0,C 180,E1 18481.307,E2 18481.307} C_VEL
LIN {X 0,Y 424.48,Z 399.245,A -85,B 0,C 180,E1 18480.809,E2 18480.809} C_VEL
LIN {X 0,Y 428.03,Z 403.647,A -85,B 0,C 180,E1 18479.928,E2 18479.928} C_VEL
LIN {X 0,Y 438.656,Z 417.375,A -85,B 0,C 180,E1 18477.463,E2 18477.463} C_VEL
LIN {X 0,Y 449.275,Z 431.522,A -85,B 0,C 180,E1 18475.221,E2 18475.221} C_VEL
LIN {X 0,Y 461.055,Z 448.275,A -85,B 0,C 180,E1 18472.922,E2 18472.922} C_VEL
LIN {X 0,Y 454.578,Z 616.417,A -85,B 0,C 180,E1 18469.83,E2 18469.83} C_VEL
LIN {X 0,Y 453.613,Z 624.115,A -85,B 0,C 180,E1 18469.784,E2 18469.784} C_VEL
LIN {X 0,Y 448.599,Z 644.7,A -85,B 0,C 180,E1 18469.994,E2 18469.994} C_VEL
LIN {X 0,Y 447.846,Z 651.305,A -85,B 0,C 180,E1 18469.943,E2 18469.943} C_VEL
LIN {X 0,Y 445.217,Z 715.801,A -85,B 0,C 180,E1 18468.732,E2 18468.732} C_VEL
LIN {X 0,Y 443.32,Z 738.58,A -85,B 0,C 180,E1 18468.1,E2 18468.1} C_VEL
LIN {X 0,Y 440.883,Z 761.401,A -85,B 0,C 180,E1 18467.244,E2 18467.244} C_VEL
LIN {X 0,Y 438.223,Z 781.117,A -85,B 0,C 180,E1 18466.294,E2 18466.294} C_VEL
LIN {X 0,Y 434.957,Z 802.296,A -85,B 0,C 180,E1 18465.051,E2 18465.051} C_VEL
LIN {X 0,Y 431.49,Z 821.664,A -85,B 0,C 180,E1 18463.667,E2 18463.667} C_VEL
LIN {X 0,Y 427.66,Z 841.361,A -85,B 0,C 180,E1 18462.005,E2 18462.005} C_VEL
LIN {X 0,Y 423.828,Z 859.504,A -85,B 0,C 180,E1 18460.187,E2 18460.187} C_VEL
LIN {X 0,Y 419.62,Z 878.63,A -85,B 0,C 180,E1 18457.939,E2 18457.939} C_VEL
LIN {X 0,Y 415.855,Z 895.241,A -85,B 0,C 180,E1 18455.653,E2 18455.653} C_VEL
LIN {X 0,Y 412.37,Z 910.506,A -85,B 0,C 180,E1 18453.193,E2 18453.193} C_VEL
LIN {X 0,Y 409.229,Z 924.704,A -85,B 0,C 180,E1 18450.556,E2 18450.556} C_VEL
LIN {X 0,Y 406.505,Z 937.556,A -85,B 0,C 180,E1 18447.74,E2 18447.74} C_VEL
LIN {X 0,Y 404.261,Z 949.334,A -85,B 0,C 180,E1 18444.745,E2 18444.745} C_VEL
LIN {X 0,Y 402.554,Z 959.261,A -85,B 0,C 180,E1 18441.713,E2 18441.713} C_VEL
LIN {X 0,Y 401.252,Z 968.483,A -85,B 0,C 180,E1 18438.324,E2 18438.324} C_VEL
LIN {X 0,Y 400.498,Z 975.536,A -85,B 0,C 180,E1 18435.095,E2 18435.095} C_VEL
LIN {X 0,Y 400.114,Z 981.134,A -85,B 0,C 180,E1 18431.733,E2 18431.733} C_VEL
LIN {X 0,Y 399.959,Z 984.804,A -85,B 0,C 180,E1 18428.59,E2 18428.59} C_VEL
LIN {X 0,Y 399.915,Z 987.163,A -85,B 0,C 180,E1 18425.318,E2 18425.318} C_VEL
LIN {X 0,Y 399.898,Z 987.997,A -85,B 0,C 180,E1 18422.265,E2 18422.265} C_VEL
LIN {X 0,Y 399.917,Z 987.419,A -85,B 0,C 180,E1 18419.164,E2 18419.164} C_VEL
LIN {X 0,Y 399.918,Z 985.411,A -85,B 0,C 180,E1 18415.938,E2 18415.938} C_VEL
LIN {X 0,Y 400.056,Z 981.95,A -85,B 0,C 180,E1 18412.78,E2 18412.78} C_VEL
LIN {X 0,Y 400.401,Z 976.829,A -85,B 0,C 180,E1 18409.511,E2 18409.511} C_VEL
LIN {X 0,Y 401.054,Z 970.243,A -85,B 0,C 180,E1 18406.303,E2 18406.303} C_VEL
LIN {X 0,Y 402.182,Z 961.868,A -85,B 0,C 180,E1 18403.033,E2 18403.033} C_VEL
LIN {X 0,Y 403.781,Z 951.946,A -85,B 0,C 180,E1 18399.893,E2 18399.893} C_VEL
LIN {X 0,Y 406.029,Z 940.193,A -85,B 0,C 180,E1 18396.756,E2 18396.756} C_VEL
LIN {X 0,Y 408.489,Z 928.425,A -85,B 0,C 180,E1 18394.093,E2 18394.093} C_VEL
LIN {X 0,Y 411.872,Z 913.149,A -85,B 0,C 180,E1 18391.137,E2 18391.137} C_VEL
LIN {X 0,Y 415.383,Z 897.959,A -85,B 0,C 180,E1 18388.621,E2 18388.621} C_VEL
LIN {X 0,Y 419.196,Z 881.116,A -85,B 0,C 180,E1 18386.251,E2 18386.251} C_VEL
LIN {X 0,Y 423.156,Z 863.647,A -85,B 0,C 180,E1 18384.128,E2 18384.128} C_VEL
LIN {X 0,Y 426.904,Z 845.914,A -85,B 0,C 180,E1 18382.299,E2 18382.299} C_VEL
LIN {X 0,Y 430.972,Z 825.583,A -85,B 0,C 180,E1 18380.508,E2 18380.508} C_VEL
LIN {X 0,Y 434.509,Z 806.061,A -85,B 0,C 180,E1 18379.073,E2 18379.073} C_VEL
LIN {X 0,Y 438.036,Z 784.157,A -85,B 0,C 180,E1 18377.742,E2 18377.742} C_VEL
LIN {X 0,Y 440.713,Z 764.653,A -85,B 0,C 180,E1 18376.777,E2 18376.777} C_VEL
LIN {X 0,Y 443.313,Z 741.353,A -85,B 0,C 180,E1 18375.87,E2 18375.87} C_VEL
LIN {X 0,Y 445.059,Z 721.056,A -85,B 0,C 180,E1 18375.281,E2 18375.281} C_VEL
LIN {X 0,Y 446.646,Z 689.481,A -85,B 0,C 180,E1 18374.639,E2 18374.639} C_VEL
LIN {X 0,Y 455.147,Z 488.509,A -85,B 0,C 180,E1 18370.873,E2 18370.873} C_VEL
LIN {X 0,Y 456.704,Z 452.49,A -85,B 0,C 180,E1 18370.167,E2 18370.167} C_VEL
LIN {X 0,Y 446.765,Z 437.56,A -85,B 0,C 180,E1 18367.944,E2 18367.944} C_VEL
LIN {X 0,Y 438.489,Z 426.305,A -85,B 0,C 180,E1 18365.89,E2 18365.89} C_VEL
LIN {X 0,Y 434.901,Z 421.556,A -85,B 0,C 180,E1 18364.913,E2 18364.913} C_VEL
LIN {X 0,Y 431.44,Z 417.044,A -85,B 0,C 180,E1 18363.921,E2 18363.921} C_VEL
LIN {X 0,Y 427.415,Z 411.882,A -85,B 0,C 180,E1 18362.665,E2 18362.665} C_VEL
LIN {X 0,Y 424,Z 407.593,A -85,B 0,C 180,E1 18361.529,E2 18361.529} C_VEL
LIN {X 0,Y 422.734,Z 406.183,A -85,B 0,C 180,E1 18361.085,E2 18361.085} C_VEL
LIN {X 0,Y 419.601,Z 402.475,A -85,B 0,C 180,E1 18359.898,E2 18359.898} C_VEL
LIN {X 0,Y 418.538,Z 400.723,A -85,B 0,C 180,E1 18359.453,E2 18359.453} C_VEL
LIN {X 0,Y 415.36,Z 397.971,A -85,B 0,C 180,E1 18358.138,E2 18358.138} C_VEL
LIN {X 0,Y 413.322,Z 394.474,A -85,B 0,C 180,E1 18357.089,E2 18357.089} C_VEL
LIN {X 0,Y 409.764,Z 391.924,A -85,B 0,C 180,E1 18355.242,E2 18355.242} C_VEL
LIN {X 0,Y 408.023,Z 388.702,A -85,B 0,C 180,E1 18353.987,E2 18353.987} C_VEL
LIN {X 0,Y 406.335,Z 387.426,A -85,B 0,C 180,E1 18352.791,E2 18352.791} C_VEL
LIN {X 0,Y 402.615,Z 384.229,A -85,B 0,C 180,E1 18347.96,E2 18347.96} C_VEL
LIN {X 0,Y 402.389,Z 383.868,A -85,B 0,C 180,E1 18345.613,E2 18345.613} C_VEL
LIN {X 0,Y 403.52,Z 385.443,A -85,B 0,C 180,E1 18342.554,E2 18342.554} C_VEL
LIN {X 0,Y 407.849,Z 388.405,A -85,B 0,C 180,E1 18338.576,E2 18338.576} C_VEL
LIN {X 0,Y 409.9,Z 392.137,A -85,B 0,C 180,E1 18337.104,E2 18337.104} C_VEL
LIN {X 0,Y 413.568,Z 394.906,A -85,B 0,C 180,E1 18335.2,E2 18335.2} C_VEL
LIN {X 0,Y 415.908,Z 398.701,A -85,B 0,C 180,E1 18334.054,E2 18334.054} C_VEL
LIN {X 0,Y 418.551,Z 401.171,A -85,B 0,C 180,E1 18332.969,E2 18332.969} C_VEL
LIN {X 0,Y 422.898,Z 406.972,A -85,B 0,C 180,E1 18331.28,E2 18331.28} C_VEL
LIN {X 0,Y 426.865,Z 412.226,A -85,B 0,C 180,E1 18329.917,E2 18329.917} C_VEL
LIN {X 0,Y 433.167,Z 420.875,A -85,B 0,C 180,E1 18327.974,E2 18327.974} C_VEL
LIN {X 0,Y 440.649,Z 432,A -85,B 0,C 180,E1 18325.913,E2 18325.913} C_VEL
LIN {X 0,Y 448.487,Z 444.204,A -85,B 0,C 180,E1 18323.985,E2 18323.985} C_VEL
LIN {X 0,Y 456.796,Z 458.138,A -85,B 0,C 180,E1 18322.123,E2 18322.123} C_VEL
LIN {X 0,Y 448.56,Z 649.793,A -85,B 0,C 180,E1 18318.509,E2 18318.509} C_VEL
LIN {X 0,Y 444.948,Z 737.873,A -85,B 0,C 180,E1 18316.852,E2 18316.852} C_VEL
LIN {X 0,Y 442.862,Z 761.387,A -85,B 0,C 180,E1 18316.221,E2 18316.221} C_VEL
LIN {X 0,Y 440.304,Z 784.09,A -85,B 0,C 180,E1 18315.394,E2 18315.394} C_VEL
LIN {X 0,Y 437.37,Z 805.178,A -85,B 0,C 180,E1 18314.393,E2 18314.393} C_VEL
LIN {X 0,Y 433.786,Z 827.901,A -85,B 0,C 180,E1 18313.058,E2 18313.058} C_VEL
LIN {X 0,Y 430.436,Z 846.66,A -85,B 0,C 180,E1 18311.725,E2 18311.725} C_VEL
LIN {X 0,Y 426.302,Z 868.054,A -85,B 0,C 180,E1 18309.92,E2 18309.92} C_VEL
LIN {X 0,Y 422.509,Z 886.564,A -85,B 0,C 180,E1 18308.075,E2 18308.075} C_VEL
LIN {X 0,Y 418.629,Z 904.852,A -85,B 0,C 180,E1 18305.937,E2 18305.937} C_VEL
LIN {X 0,Y 415.001,Z 921.769,A -85,B 0,C 180,E1 18303.655,E2 18303.655} C_VEL
LIN {X 0,Y 411.621,Z 937.567,A -85,B 0,C 180,E1 18301.161,E2 18301.161} C_VEL
LIN {X 0,Y 408.614,Z 952.267,A -85,B 0,C 180,E1 18298.503,E2 18298.503} C_VEL
LIN {X 0,Y 406.028,Z 965.545,A -85,B 0,C 180,E1 18295.673,E2 18295.673} C_VEL
LIN {X 0,Y 403.942,Z 977.555,A -85,B 0,C 180,E1 18292.718,E2 18292.718} C_VEL
LIN {X 0,Y 402.377,Z 987.677,A -85,B 0,C 180,E1 18289.755,E2 18289.755} C_VEL
LIN {X 0,Y 401.215,Z 997.006,A -85,B 0,C 180,E1 18286.509,E2 18286.509} C_VEL
LIN {X 0,Y 400.546,Z 1003.83,A -85,B 0,C 180,E1 18283.575,E2 18283.575} C_VEL
LIN {X 0,Y 400.123,Z 1009.775,A -85,B 0,C 180,E1 18280.369,E2 18280.369} C_VEL
LIN {X 0,Y 399.953,Z 1013.679,A -85,B 0,C 180,E1 18277.474,E2 18277.474} C_VEL
LIN {X 0,Y 399.909,Z 1016.371,A -85,B 0,C 180,E1 18274.593,E2 18274.593} C_VEL
LIN {X 0,Y 399.906,Z 1017.778,A -85,B 0,C 180,E1 18271.437,E2 18271.437} C_VEL
LIN {X 0,Y 399.903,Z 1017.802,A -85,B 0,C 180,E1 18268.715,E2 18268.715} C_VEL
LIN {X 0,Y 399.909,Z 1016.494,A -85,B 0,C 180,E1 18265.559,E2 18265.559} C_VEL
LIN {X 0,Y 399.944,Z 1013.857,A -85,B 0,C 180,E1 18262.68,E2 18262.68} C_VEL
LIN {X 0,Y 400.095,Z 1010.228,A -85,B 0,C 180,E1 18259.93,E2 18259.93} C_VEL
LIN {X 0,Y 400.522,Z 1004.195,A -85,B 0,C 180,E1 18256.581,E2 18256.581} C_VEL
LIN {X 0,Y 401.176,Z 997.442,A -85,B 0,C 180,E1 18253.644,E2 18253.644} C_VEL
LIN {X 0,Y 402.337,Z 988.17,A -85,B 0,C 180,E1 18250.365,E2 18250.365} C_VEL
LIN {X 0,Y 403.865,Z 978.255,A -85,B 0,C 180,E1 18247.433,E2 18247.433} C_VEL
LIN {X 0,Y 405.94,Z 966.412,A -85,B 0,C 180,E1 18244.472,E2 18244.472} C_VEL
LIN {X 0,Y 408.497,Z 953.348,A -85,B 0,C 180,E1 18241.657,E2 18241.657} C_VEL
LIN {X 0,Y 411.488,Z 938.9,A -85,B 0,C 180,E1 18239,E2 18239} C_VEL
LIN {X 0,Y 414.871,Z 923.316,A -85,B 0,C 180,E1 18236.498,E2 18236.498} C_VEL
LIN {X 0,Y 418.535,Z 906.368,A -85,B 0,C 180,E1 18234.183,E2 18234.183} C_VEL
LIN {X 0,Y 422.504,Z 887.937,A -85,B 0,C 180,E1 18232.002,E2 18232.002} C_VEL
LIN {X 0,Y 426.375,Z 869.12,A -85,B 0,C 180,E1 18230.114,E2 18230.114} C_VEL
LIN {X 0,Y 430.544,Z 847.731,A -85,B 0,C 180,E1 18228.299,E2 18228.299} C_VEL
LIN {X 0,Y 433.93,Z 828.759,A -85,B 0,C 180,E1 18226.948,E2 18226.948} C_VEL
LIN {X 0,Y 437.457,Z 806.334,A -85,B 0,C 180,E1 18225.629,E2 18225.629} C_VEL
LIN {X 0,Y 440.466,Z 784.482,A -85,B 0,C 180,E1 18224.593,E2 18224.593} C_VEL
LIN {X 0,Y 442.965,Z 761.644,A -85,B 0,C 180,E1 18223.769,E2 18223.769} C_VEL
LIN {X 0,Y 444.973,Z 738.112,A -85,B 0,C 180,E1 18223.148,E2 18223.148} C_VEL
LIN {X 0,Y 449.075,Z 633.209,A -85,B 0,C 180,E1 18221.2,E2 18221.2} C_VEL
LIN {X 0,Y 456.077,Z 458.195,A -85,B 0,C 180,E1 18217.947,E2 18217.947} C_VEL
LIN {X 0,Y 444.673,Z 440.456,A -85,B 0,C 180,E1 18215.617,E2 18215.617} C_VEL
LIN {X 0,Y 433.142,Z 423.638,A -85,B 0,C 180,E1 18213.048,E2 18213.048} C_VEL
LIN {X 0,Y 424.388,Z 411.858,A -85,B 0,C 180,E1 18210.943,E2 18210.943} C_VEL
LIN {X 0,Y 417.372,Z 402.465,A -85,B 0,C 180,E1 18209.098,E2 18209.098} C_VEL
LIN {X 0,Y 413.479,Z 397.45,A -85,B 0,C 180,E1 18208.016,E2 18208.016} C_VEL
LIN {X 0,Y 409.99,Z 392.863,A -85,B 0,C 180,E1 18207.014,E2 18207.014} C_VEL
LIN {X 0,Y 405.936,Z 388.073,A -85,B 0,C 180,E1 18205.807,E2 18205.807} C_VEL
LIN {X 0,Y 404.587,Z 386.477,A -85,B 0,C 180,E1 18205.389,E2 18205.389} C_VEL
LIN {X 0,Y 402.115,Z 383.43,A -85,B 0,C 180,E1 18204.534,E2 18204.534} C_VEL
LIN {X 0,Y 401.496,Z 381.211,A -85,B 0,C 180,E1 18203.87,E2 18203.87} C_VEL
LIN {X 0,Y 401.447,Z 381.032,A -85,B 0,C 180,E1 18200.102,E2 18200.102} C_VEL
LIN {X 0,Y 401.433,Z 381.045,A -85,B 0,C 180,E1 18196.346,E2 18196.346} C_VEL
LIN {X 0,Y 401.433,Z 381.037,A -85,B 0,C 180,E1 18192.512,E2 18192.512} C_VEL
LIN {X 0,Y 401.438,Z 381.029,A -85,B 0,C 180,E1 18188.594,E2 18188.594} C_VEL
LIN {X 0,Y 401.46,Z 381.03,A -85,B 0,C 180,E1 18184.857,E2 18184.857} C_VEL
LIN {X 0,Y 401.487,Z 381.033,A -85,B 0,C 180,E1 18180.998,E2 18180.998} C_VEL
LIN {X 0,Y 401.486,Z 381.038,A -85,B 0,C 180,E1 18177.002,E2 18177.002} C_VEL
LIN {X 0,Y 401.495,Z 381.029,A -85,B 0,C 180,E1 18172.99,E2 18172.99} C_VEL
LIN {X 0,Y 401.477,Z 381.028,A -85,B 0,C 180,E1 18169.089,E2 18169.089} C_VEL
LIN {X 0,Y 401.459,Z 381.028,A -85,B 0,C 180,E1 18165.283,E2 18165.283} C_VEL
LIN {X 0,Y 401.455,Z 381.027,A -85,B 0,C 180,E1 18161.409,E2 18161.409} C_VEL
LIN {X 0,Y 401.458,Z 381.033,A -85,B 0,C 180,E1 18157.446,E2 18157.446} C_VEL
LIN {X 0,Y 401.463,Z 381.039,A -85,B 0,C 180,E1 18153.524,E2 18153.524} C_VEL
LIN {X 0,Y 401.482,Z 381.037,A -85,B 0,C 180,E1 18149.776,E2 18149.776} C_VEL
LIN {X 0,Y 401.496,Z 381.03,A -85,B 0,C 180,E1 18145.921,E2 18145.921} C_VEL
LIN {X 0,Y 401.506,Z 381.023,A -85,B 0,C 180,E1 18141.889,E2 18141.889} C_VEL
LIN {X 0,Y 401.507,Z 381.028,A -85,B 0,C 180,E1 18137.902,E2 18137.902} C_VEL
LIN {X 0,Y 401.499,Z 381.03,A -85,B 0,C 180,E1 18133.969,E2 18133.969} C_VEL
LIN {X 0,Y 401.498,Z 381.025,A -85,B 0,C 180,E1 18129.971,E2 18129.971} C_VEL
LIN {X 0,Y 401.528,Z 381.26,A -85,B 0,C 180,E1 18127.229,E2 18127.229} C_VEL
LIN {X 0,Y 401.846,Z 382.625,A -85,B 0,C 180,E1 18126.838,E2 18126.838} C_VEL
LIN {X 0,Y 403.688,Z 385.63,A -85,B 0,C 180,E1 18126.212,E2 18126.212} C_VEL
LIN {X 0,Y 406.651,Z 387.879,A -85,B 0,C 180,E1 18125.343,E2 18125.343} C_VEL
LIN {X 0,Y 408.905,Z 391.518,A -85,B 0,C 180,E1 18124.632,E2 18124.632} C_VEL
LIN {X 0,Y 411.725,Z 394.059,A -85,B 0,C 180,E1 18123.845,E2 18123.845} C_VEL
LIN {X 0,Y 414.613,Z 398.136,A -85,B 0,C 180,E1 18123.019,E2 18123.019} C_VEL
LIN {X 0,Y 416.775,Z 400.344,A -85,B 0,C 180,E1 18122.449,E2 18122.449} C_VEL
LIN {X 0,Y 420.248,Z 404.693,A -85,B 0,C 180,E1 18121.537,E2 18121.537} C_VEL
LIN {X 0,Y 422.075,Z 406.927,A -85,B 0,C 180,E1 18121.072,E2 18121.072} C_VEL
LIN {X 0,Y 426.762,Z 412.862,A -85,B 0,C 180,E1 18119.902,E2 18119.902} C_VEL
LIN {X 0,Y 434.775,Z 423.113,A -85,B 0,C 180,E1 18118.017,E2 18118.017} C_VEL
LIN {X 0,Y 445.965,Z 438.219,A -85,B 0,C 180,E1 18115.597,E2 18115.597} C_VEL
LIN {X 0,Y 455.798,Z 452.326,A -85,B 0,C 180,E1 18113.628,E2 18113.628} C_VEL
LIN {X 0,Y 447.846,Z 651.305,A -85,B 0,C 180,E1 18109.943,E2 18109.943} C_VEL
LIN {X 0,Y 446.884,Z 659.001,A -85,B 0,C 180,E1 18109.895,E2 18109.895} C_VEL
LIN {X 0,Y 441.837,Z 679.577,A -85,B 0,C 180,E1 18110.111,E2 18110.111} C_VEL
LIN {X 0,Y 441.065,Z 686.182,A -85,B 0,C 180,E1 18110.061,E2 18110.061} C_VEL
LIN {X 0,Y 439.406,Z 719.452,A -85,B 0,C 180,E1 18109.394,E2 18109.394} C_VEL
LIN {X 0,Y 437.545,Z 740.579,A -85,B 0,C 180,E1 18108.787,E2 18108.787} C_VEL
LIN {X 0,Y 434.832,Z 764.136,A -85,B 0,C 180,E1 18107.872,E2 18107.872} C_VEL
LIN {X 0,Y 432.168,Z 782.953,A -85,B 0,C 180,E1 18106.944,E2 18106.944} C_VEL
LIN {X 0,Y 428.579,Z 804.754,A -85,B 0,C 180,E1 18105.627,E2 18105.627} C_VEL
LIN {X 0,Y 425.151,Z 823.083,A -85,B 0,C 180,E1 18104.291,E2 18104.291} C_VEL
LIN {X 0,Y 420.699,Z 844.655,A -85,B 0,C 180,E1 18102.416,E2 18102.416} C_VEL
LIN {X 0,Y 416.636,Z 863.159,A -85,B 0,C 180,E1 18100.504,E2 18100.504} C_VEL
LIN {X 0,Y 412.495,Z 880.733,A -85,B 0,C 180,E1 18098.358,E2 18098.358} C_VEL
LIN {X 0,Y 408.588,Z 897.189,A -85,B 0,C 180,E1 18096.036,E2 18096.036} C_VEL
LIN {X 0,Y 404.943,Z 912.222,A -85,B 0,C 180,E1 18093.535,E2 18093.535} C_VEL
LIN {X 0,Y 401.662,Z 926.243,A -85,B 0,C 180,E1 18090.851,E2 18090.851} C_VEL
LIN {X 0,Y 398.813,Z 938.935,A -85,B 0,C 180,E1 18087.984,E2 18087.984} C_VEL
LIN {X 0,Y 396.251,Z 951.499,A -85,B 0,C 180,E1 18084.639,E2 18084.639} C_VEL
LIN {X 0,Y 394.605,Z 960.793,A -85,B 0,C 180,E1 18081.692,E2 18081.692} C_VEL
LIN {X 0,Y 393.321,Z 969.339,A -85,B 0,C 180,E1 18078.411,E2 18078.411} C_VEL
LIN {X 0,Y 392.525,Z 976.327,A -85,B 0,C 180,E1 18075.088,E2 18075.088} C_VEL
LIN {X 0,Y 392.13,Z 981.696,A -85,B 0,C 180,E1 18071.718,E2 18071.718} C_VEL
LIN {X 0,Y 391.962,Z 985.375,A -85,B 0,C 180,E1 18068.445,E2 18068.445} C_VEL
LIN {X 0,Y 391.92,Z 987.582,A -85,B 0,C 180,E1 18065.102,E2 18065.102} C_VEL
LIN {X 0,Y 391.91,Z 988.309,A -85,B 0,C 180,E1 18061.833,E2 18061.833} C_VEL
LIN {X 0,Y 391.917,Z 987.518,A -85,B 0,C 180,E1 18058.634,E2 18058.634} C_VEL
LIN {X 0,Y 391.96,Z 985.265,A -85,B 0,C 180,E1 18055.326,E2 18055.326} C_VEL
LIN {X 0,Y 392.129,Z 981.576,A -85,B 0,C 180,E1 18052.08,E2 18052.08} C_VEL
LIN {X 0,Y 392.552,Z 976.189,A -85,B 0,C 180,E1 18048.712,E2 18048.712} C_VEL
LIN {X 0,Y 393.351,Z 969.296,A -85,B 0,C 180,E1 18045.443,E2 18045.443} C_VEL
LIN {X 0,Y 394.74,Z 960.161,A -85,B 0,C 180,E1 18041.968,E2 18041.968} C_VEL
LIN {X 0,Y 396.541,Z 950.381,A -85,B 0,C 180,E1 18038.892,E2 18038.892} C_VEL
LIN {X 0,Y 398.956,Z 938.661,A -85,B 0,C 180,E1 18035.811,E2 18035.811} C_VEL
LIN {X 0,Y 401.786,Z 926.222,A -85,B 0,C 180,E1 18032.999,E2 18032.999} C_VEL
LIN {X 0,Y 405.215,Z 911.666,A -85,B 0,C 180,E1 18030.224,E2 18030.224} C_VEL
LIN {X 0,Y 409.125,Z 895.559,A -85,B 0,C 180,E1 18027.581,E2 18027.581} C_VEL
LIN {X 0,Y 412.92,Z 879.843,A -85,B 0,C 180,E1 18025.379,E2 18025.379} C_VEL
LIN {X 0,Y 417.388,Z 860.714,A -85,B 0,C 180,E1 18023.087,E2 18023.087} C_VEL
LIN {X 0,Y 421.512,Z 842.296,A -85,B 0,C 180,E1 18021.21,E2 18021.21} C_VEL
LIN {X 0,Y 425.488,Z 822.901,A -85,B 0,C 180,E1 18019.55,E2 18019.55} C_VEL
LIN {X 0,Y 429.232,Z 803.108,A -85,B 0,C 180,E1 18018.115,E2 18018.115} C_VEL
LIN {X 0,Y 432.604,Z 782.38,A -85,B 0,C 180,E1 18016.884,E2 18016.884} C_VEL
LIN {X 0,Y 435.557,Z 761.588,A -85,B 0,C 180,E1 18015.871,E2 18015.871} C_VEL
LIN {X 0,Y 438.045,Z 738.97,A -85,B 0,C 180,E1 18015.023,E2 18015.023} C_VEL
LIN {X 0,Y 440.005,Z 716.1,A -85,B 0,C 180,E1 18014.39,E2 18014.39} C_VEL
LIN {X 0,Y 445.363,Z 594.997,A -85,B 0,C 180,E1 18012.089,E2 18012.089} C_VEL
LIN {X 0,Y 451.786,Z 456.543,A -85,B 0,C 180,E1 18009.426,E2 18009.426} C_VEL
LIN {X 0,Y 442.655,Z 442.919,A -85,B 0,C 180,E1 18007.3,E2 18007.3} C_VEL
LIN {X 0,Y 435.349,Z 432.715,A -85,B 0,C 180,E1 18005.404,E2 18005.404} C_VEL
LIN {X 0,Y 429.224,Z 424.446,A -85,B 0,C 180,E1 18003.64,E2 18003.64} C_VEL
LIN {X 0,Y 424.901,Z 418.93,A -85,B 0,C 180,E1 18002.259,E2 18002.259} C_VEL
LIN {X 0,Y 420.793,Z 413.695,A -85,B 0,C 180,E1 18000.817,E2 18000.817} C_VEL
LIN {X 0,Y 417.444,Z 409.677,A -85,B 0,C 180,E1 17999.52,E2 17999.52} C_VEL
LIN {X 0,Y 416.283,Z 408.081,A -85,B 0,C 180,E1 17999.037,E2 17999.037} C_VEL
LIN {X 0,Y 413.086,Z 404.797,A -85,B 0,C 180,E1 17997.608,E2 17997.608} C_VEL
LIN {X 0,Y 411.564,Z 402.132,A -85,B 0,C 180,E1 17996.797,E2 17996.797} C_VEL
LIN {X 0,Y 408.158,Z 399.476,A -85,B 0,C 180,E1 17994.941,E2 17994.941} C_VEL
LIN {X 0,Y 406.222,Z 395.91,A -85,B 0,C 180,E1 17993.499,E2 17993.499} C_VEL
LIN {X 0,Y 401.912,Z 392.777,A -85,B 0,C 180,E1 17988.957,E2 17988.957} C_VEL
LIN {X 0,Y 401.287,Z 391.703,A -85,B 0,C 180,E1 17986.161,E2 17986.161} C_VEL
LIN {X 0,Y 401.951,Z 392.849,A -85,B 0,C 180,E1 17983.378,E2 17983.378} C_VEL
